LIN {X 0,Y 503.622,Z 638.337,A -85,B 0,C 180,E1 23233.198,E2 23233.198} C_VEL
LIN {X 0,Y 501.583,Z 634.122,A -85,B 0,C 180,E1 23232.199,E2 23232.199} C_VEL
LIN {X 0,Y 499.58,Z 629.914,A -85,B 0,C 180,E1 23231.195,E2 23231.195} C_VEL
LIN {X 0,Y 498.04,Z 626.665,A -85,B 0,C 180,E1 23230.41,E2 23230.41} C_VEL
LIN {X 0,Y 497.921,Z 625.951,A -85,B 0,C 180,E1 23230.237,E2 23230.237} C_VEL
LIN {X 0,Y 497.932,Z 625.949,A -85,B 0,C 180,E1 23226.688,E2 23226.688} C_VEL
LIN {X 0,Y 497.917,Z 625.952,A -85,B 0,C 180,E1 23223.108,E2 23223.108} C_VEL
LIN {X 0,Y 497.933,Z 625.957,A -85,B 0,C 180,E1 23219.54,E2 23219.54} C_VEL
LIN {X 0,Y 497.926,Z 625.949,A -85,B 0,C 180,E1 23215.854,E2 23215.854} C_VEL
LIN {X 0,Y 497.932,Z 625.949,A -85,B 0,C 180,E1 23212.268,E2 23212.268} C_VEL
LIN {X 0,Y 497.92,Z 625.957,A -85,B 0,C 180,E1 23208.65,E2 23208.65} C_VEL
LIN {X 0,Y 497.926,Z 625.958,A -85,B 0,C 180,E1 23205.106,E2 23205.106} C_VEL
LIN {X 0,Y 497.935,Z 625.96,A -85,B 0,C 180,E1 23201.502,E2 23201.502} C_VEL
LIN {X 0,Y 497.922,Z 625.959,A -85,B 0,C 180,E1 23197.943,E2 23197.943} C_VEL
LIN {X 0,Y 497.927,Z 625.957,A -85,B 0,C 180,E1 23194.294,E2 23194.294} C_VEL
LIN {X 0,Y 497.919,Z 625.959,A -85,B 0,C 180,E1 23190.792,E2 23190.792} C_VEL
LIN {X 0,Y 497.93,Z 625.957,A -85,B 0,C 180,E1 23187.283,E2 23187.283} C_VEL
LIN {X 0,Y 497.923,Z 625.955,A -85,B 0,C 180,E1 23183.815,E2 23183.815} C_VEL
LIN {X 0,Y 497.93,Z 625.956,A -85,B 0,C 180,E1 23180.27,E2 23180.27} C_VEL
LIN {X 0,Y 497.92,Z 625.916,A -85,B 0,C 180,E1 23176.628,E2 23176.628} C_VEL
LIN {X 0,Y 497.928,Z 625.947,A -85,B 0,C 180,E1 23173.056,E2 23173.056} C_VEL
LIN {X 0,Y 497.936,Z 625.963,A -85,B 0,C 180,E1 23169.533,E2 23169.533} C_VEL
LIN {X 0,Y 497.945,Z 626.094,A -85,B 0,C 180,E1 23169.367,E2 23169.367} C_VEL
LIN {X 0,Y 507.09,Z 649.982,A -85,B 0,C 180,E1 23166.816,E2 23166.816} C_VEL
LIN {X 0,Y 513.886,Z 670.595,A -85,B 0,C 180,E1 23164.716,E2 23164.716} C_VEL
LIN {X 0,Y 516.12,Z 678.989,A -85,B 0,C 180,E1 23163.912,E2 23163.912} C_VEL
LIN {X 0,Y 514.134,Z 718.892,A -85,B 0,C 180,E1 23160.89,E2 23160.89} C_VEL
LIN {X 0,Y 511.854,Z 763.473,A -85,B 0,C 180,E1 23157.516,E2 23157.516} C_VEL
LIN {X 0,Y 509.643,Z 811.319,A -85,B 0,C 180,E1 23153.959,E2 23153.959} C_VEL
LIN {X 0,Y 508.296,Z 851.099,A -85,B 0,C 180,E1 23151.154,E2 23151.154} C_VEL
LIN {X 0,Y 509.003,Z 858.968,A -85,B 0,C 180,E1 23151.003,E2 23151.003} C_VEL
LIN {X 0,Y 506.584,Z 1020.416,A -85,B 0,C 180,E1 23148.679,E2 23148.679} C_VEL
LIN {X 0,Y 506.284,Z 1037.996,A -85,B 0,C 180,E1 23148.228,E2 23148.228} C_VEL
LIN {X 0,Y 505.713,Z 1054.181,A -85,B 0,C 180,E1 23147.607,E2 23147.607} C_VEL
LIN {X 0,Y 505.321,Z 1062.229,A -85,B 0,C 180,E1 23147.218,E2 23147.218} C_VEL
LIN {X 0,Y 503.989,Z 1069.347,A -85,B 0,C 180,E1 23146.868,E2 23146.868} C_VEL
LIN {X 0,Y 497.857,Z 1084.669,A -85,B 0,C 180,E1 23146.084,E2 23146.084} C_VEL
LIN {X 0,Y 495.985,Z 1091.125,A -85,B 0,C 180,E1 23145.643,E2 23145.643} C_VEL
LIN {X 0,Y 495.757,Z 1092.898,A -85,B 0,C 180,E1 23145.5,E2 23145.5} C_VEL
LIN {X 0,Y 494.579,Z 1106.659,A -85,B 0,C 180,E1 23144.218,E2 23144.218} C_VEL
LIN {X 0,Y 493.371,Z 1119.245,A -85,B 0,C 180,E1 23142.76,E2 23142.76} C_VEL
LIN {X 0,Y 492.214,Z 1130.691,A -85,B 0,C 180,E1 23141.125,E2 23141.125} C_VEL
LIN {X 0,Y 491.214,Z 1140.574,A -85,B 0,C 180,E1 23139.37,E2 23139.37} C_VEL
LIN {X 0,Y 490.396,Z 1148.83,A -85,B 0,C 180,E1 23137.496,E2 23137.496} C_VEL
LIN {X 0,Y 489.788,Z 1155.493,A -85,B 0,C 180,E1 23135.504,E2 23135.504} C_VEL
LIN {X 0,Y 489.392,Z 1160.26,A -85,B 0,C 180,E1 23133.512,E2 23133.512} C_VEL
LIN {X 0,Y 489.172,Z 1163.258,A -85,B 0,C 180,E1 23131.521,E2 23131.521} C_VEL
LIN {X 0,Y 489.082,Z 1164.606,A -85,B 0,C 180,E1 23129.413,E2 23129.413} C_VEL
LIN {X 0,Y 489.126,Z 1164.179,A -85,B 0,C 180,E1 23127.304,E2 23127.304} C_VEL
LIN {X 0,Y 489.319,Z 1161.943,A -85,B 0,C 180,E1 23125.193,E2 23125.193} C_VEL
LIN {X 0,Y 489.663,Z 1158.025,A -85,B 0,C 180,E1 23123.197,E2 23123.197} C_VEL
LIN {X 0,Y 490.209,Z 1152.292,A -85,B 0,C 180,E1 23121.199,E2 23121.199} C_VEL
LIN {X 0,Y 490.957,Z 1145.049,A -85,B 0,C 180,E1 23119.318,E2 23119.318} C_VEL
LIN {X 0,Y 491.891,Z 1136.305,A -85,B 0,C 180,E1 23117.555,E2 23117.555} C_VEL
LIN {X 0,Y 492.983,Z 1126.106,A -85,B 0,C 180,E1 23115.912,E2 23115.912} C_VEL
LIN {X 0,Y 494.201,Z 1114.401,A -85,B 0,C 180,E1 23114.38,E2 23114.38} C_VEL
LIN {X 0,Y 495.469,Z 1101.282,A -85,B 0,C 180,E1 23112.984,E2 23112.984} C_VEL
LIN {X 0,Y 496.686,Z 1086.899,A -85,B 0,C 180,E1 23111.756,E2 23111.756} C_VEL
LIN {X 0,Y 497.789,Z 1071.409,A -85,B 0,C 180,E1 23110.704,E2 23110.704} C_VEL
LIN {X 0,Y 498.655,Z 1055.917,A -85,B 0,C 180,E1 23109.885,E2 23109.885} C_VEL
LIN {X 0,Y 499.309,Z 1038.979,A -85,B 0,C 180,E1 23109.22,E2 23109.22} C_VEL
LIN {X 0,Y 499.63,Z 1021.423,A -85,B 0,C 180,E1 23108.762,E2 23108.762} C_VEL
LIN {X 0,Y 501.594,Z 894.511,A -85,B 0,C 180,E1 23106.898,E2 23106.898} C_VEL
LIN {X 0,Y 502.065,Z 856.472,A -85,B 0,C 180,E1 23106.339,E2 23106.339} C_VEL
LIN {X 0,Y 501.456,Z 851.589,A -85,B 0,C 180,E1 23106.218,E2 23106.218} C_VEL
LIN {X 0,Y 503.183,Z 807.728,A -85,B 0,C 180,E1 23103.058,E2 23103.058} C_VEL
LIN {X 0,Y 505.515,Z 762.418,A -85,B 0,C 180,E1 23099.643,E2 23099.643} C_VEL
LIN {X 0,Y 508.171,Z 714.262,A -85,B 0,C 180,E1 23095.957,E2 23095.957} C_VEL
LIN {X 0,Y 509.871,Z 682.308,A -85,B 0,C 180,E1 23093.518,E2 23093.518} C_VEL
LIN {X 0,Y 503.228,Z 661.234,A -85,B 0,C 180,E1 23091.341,E2 23091.341} C_VEL
LIN {X 0,Y 495.525,Z 640.587,A -85,B 0,C 180,E1 23089.085,E2 23089.085} C_VEL
LIN {X 0,Y 490.002,Z 627.063,A -85,B 0,C 180,E1 23087.55,E2 23087.55} C_VEL
LIN {X 0,Y 490.019,Z 627.136,A -85,B 0,C 180,E1 23087.237,E2 23087.237} C_VEL
LIN {X 0,Y 491.489,Z 630.701,A -85,B 0,C 180,E1 23086.556,E2 23086.556} C_VEL
LIN {X 0,Y 498.257,Z 644.719,A -85,B 0,C 180,E1 23083.909,E2 23083.909} C_VEL
LIN {X 0,Y 500.365,Z 648.918,A -85,B 0,C 180,E1 23083.205,E2 23083.205} C_VEL
LIN {X 0,Y 518.762,Z 674.964,A -85,B 0,C 180,E1 23080.671,E2 23080.671} C_VEL
LIN {X 0,Y 534.168,Z 697.824,A -85,B 0,C 180,E1 23078.718,E2 23078.718} C_VEL
LIN {X 0,Y 520.026,Z 971.597,A -85,B 0,C 180,E1 23073.818,E2 23073.818} C_VEL
LIN {X 0,Y 518.593,Z 994.45,A -85,B 0,C 180,E1 23073.196,E2 23073.196} C_VEL
LIN {X 0,Y 516.689,Z 1017.478,A -85,B 0,C 180,E1 23072.37,E2 23072.37} C_VEL
LIN {X 0,Y 514.491,Z 1039.246,A -85,B 0,C 180,E1 23071.389,E2 23071.389} C_VEL
LIN {X 0,Y 512.002,Z 1059.668,A -85,B 0,C 180,E1 23070.255,E2 23070.255} C_VEL
LIN {X 0,Y 509.133,Z 1081.117,A -85,B 0,C 180,E1 23068.832,E2 23068.832} C_VEL
LIN {X 0,Y 506.332,Z 1100.244,A -85,B 0,C 180,E1 23067.331,E2 23067.331} C_VEL
LIN {X 0,Y 503.44,Z 1118.322,A -85,B 0,C 180,E1 23065.657,E2 23065.657} C_VEL
LIN {X 0,Y 500.455,Z 1136.635,A -85,B 0,C 180,E1 23063.678,E2 23063.678} C_VEL
LIN {X 0,Y 497.838,Z 1152.47,A -85,B 0,C 180,E1 23061.688,E2 23061.688} C_VEL
LIN {X 0,Y 495.417,Z 1167.155,A -85,B 0,C 180,E1 23059.516,E2 23059.516} C_VEL
LIN {X 0,Y 493.209,Z 1181.129,A -85,B 0,C 180,E1 23057.095,E2 23057.095} C_VEL
LIN {X 0,Y 491.538,Z 1192.748,A -85,B 0,C 180,E1 23054.731,E2 23054.731} C_VEL
LIN {X 0,Y 490.203,Z 1202.859,A -85,B 0,C 180,E1 23052.248,E2 23052.248} C_VEL
LIN {X 0,Y 489.216,Z 1211.985,A -85,B 0,C 180,E1 23049.529,E2 23049.529} C_VEL
LIN {X 0,Y 488.65,Z 1218.647,A -85,B 0,C 180,E1 23047.052,E2 23047.052} C_VEL
LIN {X 0,Y 488.301,Z 1223.926,A -85,B 0,C 180,E1 23044.463,E2 23044.463} C_VEL
LIN {X 0,Y 488.147,Z 1227.754,A -85,B 0,C 180,E1 23041.878,E2 23041.878} C_VEL
LIN {X 0,Y 488.091,Z 1229.852,A -85,B 0,C 180,E1 23039.413,E2 23039.413} C_VEL
LIN {X 0,Y 488.086,Z 1230.749,A -85,B 0,C 180,E1 23036.829,E2 23036.829} C_VEL
LIN {X 0,Y 488.12,Z 1230.019,A -85,B 0,C 180,E1 23034.239,E2 23034.239} C_VEL
LIN {X 0,Y 488.209,Z 1227.733,A -85,B 0,C 180,E1 23031.52,E2 23031.52} C_VEL
LIN {X 0,Y 488.421,Z 1224.179,A -85,B 0,C 180,E1 23029.024,E2 23029.024} C_VEL
LIN {X 0,Y 488.853,Z 1218.825,A -85,B 0,C 180,E1 23026.395,E2 23026.395} C_VEL
LIN {X 0,Y 489.556,Z 1212.199,A -85,B 0,C 180,E1 23023.873,E2 23023.873} C_VEL
LIN {X 0,Y 490.6,Z 1203.943,A -85,B 0,C 180,E1 23021.393,E2 23021.393} C_VEL
LIN {X 0,Y 492.129,Z 1193.445,A -85,B 0,C 180,E1 23018.798,E2 23018.798} C_VEL
LIN {X 0,Y 493.919,Z 1182.352,A -85,B 0,C 180,E1 23016.496,E2 23016.496} C_VEL
LIN {X 0,Y 496.141,Z 1169.08,A -85,B 0,C 180,E1 23014.195,E2 23014.195} C_VEL
LIN {X 0,Y 498.52,Z 1155.148,A -85,B 0,C 180,E1 23012.139,E2 23012.139} C_VEL
LIN {X 0,Y 501.101,Z 1140.099,A -85,B 0,C 180,E1 23010.228,E2 23010.228} C_VEL
LIN {X 0,Y 503.629,Z 1124.294,A -85,B 0,C 180,E1 23008.523,E2 23008.523} C_VEL
LIN {X 0,Y 506.268,Z 1106.682,A -85,B 0,C 180,E1 23006.9,E2 23006.9} C_VEL
LIN {X 0,Y 508.688,Z 1089.092,A -85,B 0,C 180,E1 23005.521,E2 23005.521} C_VEL
LIN {X 0,Y 510.84,Z 1070.657,A -85,B 0,C 180,E1 23004.318,E2 23004.318} C_VEL
LIN {X 0,Y 512.763,Z 1050.458,A -85,B 0,C 180,E1 23003.226,E2 23003.226} C_VEL
LIN {X 0,Y 514.255,Z 1030.564,A -85,B 0,C 180,E1 23002.362,E2 23002.362} C_VEL
LIN {X 0,Y 515.293,Z 1009.487,A -85,B 0,C 180,E1 23001.655,E2 23001.655} C_VEL
LIN {X 0,Y 515.797,Z 988.179,A -85,B 0,C 180,E1 23001.151,E2 23001.151} C_VEL
LIN {X 0,Y 517.226,Z 940.752,A -85,B 0,C 180,E1 23000.326,E2 23000.326} C_VEL
LIN {X 0,Y 520.642,Z 879.085,A -85,B 0,C 180,E1 22999.174,E2 22999.174} C_VEL
LIN {X 0,Y 525.552,Z 819.384,A -85,B 0,C 180,E1 22997.917,E2 22997.917} C_VEL
LIN {X 0,Y 527.75,Z 796.96,A -85,B 0,C 180,E1 22997.398,E2 22997.398} C_VEL
LIN {X 0,Y 520.311,Z 808.831,A -85,B 0,C 180,E1 22996.188,E2 22996.188} C_VEL
LIN {X 0,Y 515.367,Z 820.417,A -85,B 0,C 180,E1 22994.988,E2 22994.988} C_VEL
LIN {X 0,Y 512.446,Z 832.873,A -85,B 0,C 180,E1 22993.758,E2 22993.758} C_VEL
LIN {X 0,Y 511.546,Z 846.864,A -85,B 0,C 180,E1 22992.457,E2 22992.457} C_VEL
LIN {X 0,Y 512.945,Z 861.88,A -85,B 0,C 180,E1 22991.105,E2 22991.105} C_VEL
LIN {X 0,Y 517.01,Z 878.772,A -85,B 0,C 180,E1 22989.649,E2 22989.649} C_VEL
LIN {X 0,Y 522.772,Z 895.04,A -85,B 0,C 180,E1 22988.353,E2 22988.353} C_VEL
LIN {X 0,Y 530.728,Z 911.414,A -85,B 0,C 180,E1 22987.081,E2 22987.081} C_VEL
LIN {X 0,Y 524.079,Z 932.845,A -85,B 0,C 180,E1 22987.102,E2 22987.102} C_VEL
LIN {X 0,Y 519.267,Z 950.939,A -85,B 0,C 180,E1 22986.962,E2 22986.962} C_VEL
LIN {X 0,Y 515.69,Z 968.825,A -85,B 0,C 180,E1 22986.636,E2 22986.636} C_VEL
LIN {X 0,Y 513.389,Z 987.439,A -85,B 0,C 180,E1 22986.107,E2 22986.107} C_VEL
LIN {X 0,Y 509.621,Z 1023.418,A -85,B 0,C 180,E1 22984.852,E2 22984.852} C_VEL
LIN {X 0,Y 506.382,Z 1054.848,A -85,B 0,C 180,E1 22983.532,E2 22983.532} C_VEL
LIN {X 0,Y 503.423,Z 1085.64,A -85,B 0,C 180,E1 22981.994,E2 22981.994} C_VEL
LIN {X 0,Y 500.875,Z 1113.859,A -85,B 0,C 180,E1 22980.337,E2 22980.337} C_VEL
LIN {X 0,Y 498.595,Z 1139.721,A -85,B 0,C 180,E1 22978.575,E2 22978.575} C_VEL
LIN {X 0,Y 496.528,Z 1163.782,A -85,B 0,C 180,E1 22976.685,E2 22976.685} C_VEL
LIN {X 0,Y 494.62,Z 1185.737,A -85,B 0,C 180,E1 22974.675,E2 22974.675} C_VEL
LIN {X 0,Y 493.041,Z 1204.656,A -85,B 0,C 180,E1 22972.665,E2 22972.665} C_VEL
LIN {X 0,Y 491.658,Z 1221.239,A -85,B 0,C 180,E1 22970.601,E2 22970.601} C_VEL
LIN {X 0,Y 490.58,Z 1235.432,A -85,B 0,C 180,E1 22968.541,E2 22968.541} C_VEL
LIN {X 0,Y 489.663,Z 1248.183,A -85,B 0,C 180,E1 22966.369,E2 22966.369} C_VEL
LIN {X 0,Y 488.999,Z 1258.805,A -85,B 0,C 180,E1 22964.205,E2 22964.205} C_VEL
LIN {X 0,Y 488.554,Z 1267.998,A -85,B 0,C 180,E1 22961.931,E2 22961.931} C_VEL
LIN {X 0,Y 488.252,Z 1275.736,A -85,B 0,C 180,E1 22959.55,E2 22959.55} C_VEL
LIN {X 0,Y 488.122,Z 1281.616,A -85,B 0,C 180,E1 22957.18,E2 22957.18} C_VEL
LIN {X 0,Y 488.072,Z 1285.747,A -85,B 0,C 180,E1 22954.82,E2 22954.82} C_VEL
LIN {X 0,Y 488.064,Z 1288.404,A -85,B 0,C 180,E1 22952.35,E2 22952.35} C_VEL
LIN {X 0,Y 488.082,Z 1289.345,A -85,B 0,C 180,E1 22950.002,E2 22950.002} C_VEL
LIN {X 0,Y 488.042,Z 1288.685,A -85,B 0,C 180,E1 22947.536,E2 22947.536} C_VEL
LIN {X 0,Y 488.033,Z 1286.434,A -85,B 0,C 180,E1 22945.065,E2 22945.065} C_VEL
LIN {X 0,Y 488.072,Z 1282.457,A -85,B 0,C 180,E1 22942.548,E2 22942.548} C_VEL
LIN {X 0,Y 488.237,Z 1276.355,A -85,B 0,C 180,E1 22939.858,E2 22939.858} C_VEL
LIN {X 0,Y 488.608,Z 1268.875,A -85,B 0,C 180,E1 22937.354,E2 22937.354} C_VEL
LIN {X 0,Y 489.31,Z 1258.996,A -85,B 0,C 180,E1 22934.692,E2 22934.692} C_VEL
LIN {X 0,Y 490.393,Z 1247.083,A -85,B 0,C 180,E1 22932.07,E2 22932.07} C_VEL
LIN {X 0,Y 491.81,Z 1234.099,A -85,B 0,C 180,E1 22929.658,E2 22929.658} C_VEL
LIN {X 0,Y 493.701,Z 1218.912,A -85,B 0,C 180,E1 22927.245,E2 22927.245} C_VEL
LIN {X 0,Y 496.134,Z 1201.151,A -85,B 0,C 180,E1 22924.836,E2 22924.836} C_VEL
LIN {X 0,Y 498.818,Z 1182.632,A -85,B 0,C 180,E1 22922.677,E2 22922.677} C_VEL
LIN {X 0,Y 501.889,Z 1162.559,A -85,B 0,C 180,E1 22920.656,E2 22920.656} C_VEL
LIN {X 0,Y 505.491,Z 1139.288,A -85,B 0,C 180,E1 22918.655,E2 22918.655} C_VEL
LIN {X 0,Y 508.695,Z 1118.909,A -85,B 0,C 180,E1 22917.148,E2 22917.148} C_VEL
LIN {X 0,Y 512.451,Z 1094.537,A -85,B 0,C 180,E1 22915.609,E2 22915.609} C_VEL
LIN {X 0,Y 515.778,Z 1072.564,A -85,B 0,C 180,E1 22914.441,E2 22914.441} C_VEL
LIN {X 0,Y 519.332,Z 1047.797,A -85,B 0,C 180,E1 22913.358,E2 22913.358} C_VEL
LIN {X 0,Y 522.293,Z 1025.669,A -85,B 0,C 180,E1 22912.57,E2 22912.57} C_VEL
LIN {X 0,Y 525.245,Z 999.637,A -85,B 0,C 180,E1 22911.846,E2 22911.846} C_VEL
LIN {X 0,Y 527.354,Z 975.274,A -85,B 0,C 180,E1 22911.33,E2 22911.33} C_VEL
LIN {X 0,Y 530.154,Z 954.931,A -85,B 0,C 180,E1 22911.079,E2 22911.079} C_VEL
LIN {X 0,Y 532.607,Z 942.044,A -85,B 0,C 180,E1 22910.963,E2 22910.963} C_VEL
LIN {X 0,Y 536.49,Z 935.316,A -85,B 0,C 180,E1 22910.582,E2 22910.582} C_VEL
LIN {X 0,Y 529.21,Z 920.705,A -85,B 0,C 180,E1 22908.748,E2 22908.748} C_VEL
LIN {X 0,Y 523.75,Z 904.487,A -85,B 0,C 180,E1 22906.826,E2 22906.826} C_VEL
LIN {X 0,Y 520.425,Z 886.754,A -85,B 0,C 180,E1 22904.839,E2 22904.839} C_VEL
LIN {X 0,Y 519.332,Z 867.376,A -85,B 0,C 180,E1 22902.816,E2 22902.816} C_VEL
LIN {X 0,Y 520.601,Z 845.317,A -85,B 0,C 180,E1 22900.657,E2 22900.657} C_VEL
LIN {X 0,Y 525.45,Z 806.808,A -85,B 0,C 180,E1 22897.047,E2 22897.047} C_VEL
LIN {X 0,Y 530.041,Z 771.847,A -85,B 0,C 180,E1 22893.708,E2 22893.708} C_VEL
LIN {X 0,Y 534.385,Z 739.455,A -85,B 0,C 180,E1 22890.537,E2 22890.537} C_VEL
LIN {X 0,Y 535.607,Z 729.994,A -85,B 0,C 180,E1 22889.589,E2 22889.589} C_VEL
LIN {X 0,Y 527.935,Z 710.743,A -85,B 0,C 180,E1 22886.429,E2 22886.429} C_VEL
LIN {X 0,Y 520.037,Z 692,A -85,B 0,C 180,E1 22883.094,E2 22883.094} C_VEL
LIN {X 0,Y 512.802,Z 675.646,A -85,B 0,C 180,E1 22879.952,E2 22879.952} C_VEL
LIN {X 0,Y 506.279,Z 661.298,A -85,B 0,C 180,E1 22876.996,E2 22876.996} C_VEL
LIN {X 0,Y 499.858,Z 647.869,A -85,B 0,C 180,E1 22874.007,E2 22874.007} C_VEL
LIN {X 0,Y 495.726,Z 639.359,A -85,B 0,C 180,E1 22871.991,E2 22871.991} C_VEL
LIN {X 0,Y 493.67,Z 635.137,A -85,B 0,C 180,E1 22870.976,E2 22870.976} C_VEL
LIN {X 0,Y 491.719,Z 630.999,A -85,B 0,C 180,E1 22869.953,E2 22869.953} C_VEL
LIN {X 0,Y 490.138,Z 627.802,A -85,B 0,C 180,E1 22869.132,E2 22869.132} C_VEL
LIN {X 0,Y 489.988,Z 626.938,A -85,B 0,C 180,E1 22868.922,E2 22868.922} C_VEL
LIN {X 0,Y 489.995,Z 626.939,A -85,B 0,C 180,E1 22865.386,E2 22865.386} C_VEL
LIN {X 0,Y 489.994,Z 626.938,A -85,B 0,C 180,E1 22861.637,E2 22861.637} C_VEL
LIN {X 0,Y 489.979,Z 626.939,A -85,B 0,C 180,E1 22858.012,E2 22858.012} C_VEL
LIN {X 0,Y 489.989,Z 626.946,A -85,B 0,C 180,E1 22854.379,E2 22854.379} C_VEL
LIN {X 0,Y 489.984,Z 626.945,A -85,B 0,C 180,E1 22850.841,E2 22850.841} C_VEL
LIN {X 0,Y 489.992,Z 626.94,A -85,B 0,C 180,E1 22847.259,E2 22847.259} C_VEL
LIN {X 0,Y 489.984,Z 626.938,A -85,B 0,C 180,E1 22843.644,E2 22843.644} C_VEL
LIN {X 0,Y 489.991,Z 626.937,A -85,B 0,C 180,E1 22840.075,E2 22840.075} C_VEL
LIN {X 0,Y 489.989,Z 626.936,A -85,B 0,C 180,E1 22836.551,E2 22836.551} C_VEL
LIN {X 0,Y 489.98,Z 626.934,A -85,B 0,C 180,E1 22833.062,E2 22833.062} C_VEL
LIN {X 0,Y 489.985,Z 626.938,A -85,B 0,C 180,E1 22829.597,E2 22829.597} C_VEL
LIN {X 0,Y 489.996,Z 626.938,A -85,B 0,C 180,E1 22825.94,E2 22825.94} C_VEL
LIN {X 0,Y 489.997,Z 626.939,A -85,B 0,C 180,E1 22822.252,E2 22822.252} C_VEL
LIN {X 0,Y 489.985,Z 626.939,A -85,B 0,C 180,E1 22818.61,E2 22818.61} C_VEL
LIN {X 0,Y 489.981,Z 626.924,A -85,B 0,C 180,E1 22815.078,E2 22815.078} C_VEL
LIN {X 0,Y 489.998,Z 626.914,A -85,B 0,C 180,E1 22811.504,E2 22811.504} C_VEL
LIN {X 0,Y 489.986,Z 626.981,A -85,B 0,C 180,E1 22809.95,E2 22809.95} C_VEL
LIN {X 0,Y 498.827,Z 649.766,A -85,B 0,C 180,E1 22807.46,E2 22807.46} C_VEL
LIN {X 0,Y 505.699,Z 669.989,A -85,B 0,C 180,E1 22805.352,E2 22805.352} C_VEL
LIN {X 0,Y 508.926,Z 681.63,A -85,B 0,C 180,E1 22804.193,E2 22804.193} C_VEL
LIN {X 0,Y 506.912,Z 721.32,A -85,B 0,C 180,E1 22801.181,E2 22801.181} C_VEL
LIN {X 0,Y 504.446,Z 767.454,A -85,B 0,C 180,E1 22797.664,E2 22797.664} C_VEL
LIN {X 0,Y 502.253,Z 813.696,A -85,B 0,C 180,E1 22794.209,E2 22794.209} C_VEL
LIN {X 0,Y 500.918,Z 852.144,A -85,B 0,C 180,E1 22791.488,E2 22791.488} C_VEL
LIN {X 0,Y 501.594,Z 859.853,A -85,B 0,C 180,E1 22791.338,E2 22791.338} C_VEL
LIN {X 0,Y 499.074,Z 1021.09,A -85,B 0,C 180,E1 22788.985,E2 22788.985} C_VEL
LIN {X 0,Y 498.765,Z 1038.703,A -85,B 0,C 180,E1 22788.529,E2 22788.529} C_VEL
LIN {X 0,Y 498.157,Z 1055.322,A -85,B 0,C 180,E1 22787.883,E2 22787.883} C_VEL
LIN {X 0,Y 497.267,Z 1071.796,A -85,B 0,C 180,E1 22787.01,E2 22787.01} C_VEL
LIN {X 0,Y 496.21,Z 1087.141,A -85,B 0,C 180,E1 22785.963,E2 22785.963} C_VEL
LIN {X 0,Y 495.757,Z 1092.898,A -85,B 0,C 180,E1 22785.5,E2 22785.5} C_VEL
LIN {X 0,Y 494.313,Z 1099.187,A -85,B 0,C 180,E1 22784.998,E2 22784.998} C_VEL
LIN {X 0,Y 488.294,Z 1111.875,A -85,B 0,C 180,E1 22783.925,E2 22783.925} C_VEL
LIN {X 0,Y 485.952,Z 1118.163,A -85,B 0,C 180,E1 22783.24,E2 22783.24} C_VEL
LIN {X 0,Y 485.702,Z 1119.657,A -85,B 0,C 180,E1 22783.048,E2 22783.048} C_VEL
LIN {X 0,Y 484.479,Z 1131.231,A -85,B 0,C 180,E1 22781.382,E2 22781.382} C_VEL
LIN {X 0,Y 483.443,Z 1140.967,A -85,B 0,C 180,E1 22779.642,E2 22779.642} C_VEL
LIN {X 0,Y 482.619,Z 1148.928,A -85,B 0,C 180,E1 22777.857,E2 22777.857} C_VEL
LIN {X 0,Y 481.944,Z 1155.798,A -85,B 0,C 180,E1 22775.833,E2 22775.833} C_VEL
LIN {X 0,Y 481.501,Z 1160.747,A -85,B 0,C 180,E1 22773.809,E2 22773.809} C_VEL
LIN {X 0,Y 481.244,Z 1164.101,A -85,B 0,C 180,E1 22771.665,E2 22771.665} C_VEL
LIN {X 0,Y 481.141,Z 1165.539,A -85,B 0,C 180,E1 22769.522,E2 22769.522} C_VEL
LIN {X 0,Y 481.18,Z 1165.191,A -85,B 0,C 180,E1 22767.378,E2 22767.378} C_VEL
LIN {X 0,Y 481.378,Z 1163.056,A -85,B 0,C 180,E1 22765.232,E2 22765.232} C_VEL
LIN {X 0,Y 481.735,Z 1159.243,A -85,B 0,C 180,E1 22763.204,E2 22763.204} C_VEL
LIN {X 0,Y 482.299,Z 1153.599,A -85,B 0,C 180,E1 22761.174,E2 22761.174} C_VEL
LIN {X 0,Y 483.073,Z 1146.453,A -85,B 0,C 180,E1 22759.262,E2 22759.262} C_VEL
LIN {X 0,Y 484.045,Z 1137.864,A -85,B 0,C 180,E1 22757.472,E2 22757.472} C_VEL
LIN {X 0,Y 485.175,Z 1127.799,A -85,B 0,C 180,E1 22755.802,E2 22755.802} C_VEL
LIN {X 0,Y 486.426,Z 1116.308,A -85,B 0,C 180,E1 22754.255,E2 22754.255} C_VEL
LIN {X 0,Y 487.772,Z 1102.991,A -85,B 0,C 180,E1 22752.797,E2 22752.797} C_VEL
LIN {X 0,Y 489.019,Z 1089.166,A -85,B 0,C 180,E1 22751.575,E2 22751.575} C_VEL
LIN {X 0,Y 490.152,Z 1074.106,A -85,B 0,C 180,E1 22750.515,E2 22750.515} C_VEL
LIN {X 0,Y 491.113,Z 1057.858,A -85,B 0,C 180,E1 22749.624,E2 22749.624} C_VEL
LIN {X 0,Y 491.826,Z 1040.688,A -85,B 0,C 180,E1 22748.926,E2 22748.926} C_VEL
LIN {X 0,Y 492.179,Z 1023.103,A -85,B 0,C 180,E1 22748.451,E2 22748.451} C_VEL
LIN {X 0,Y 493.142,Z 956.489,A -85,B 0,C 180,E1 22747.44,E2 22747.44} C_VEL
LIN {X 0,Y 494.737,Z 857.413,A -85,B 0,C 180,E1 22745.979,E2 22745.979} C_VEL
LIN {X 0,Y 494.122,Z 852.727,A -85,B 0,C 180,E1 22745.872,E2 22745.872} C_VEL
LIN {X 0,Y 495.912,Z 808.893,A -85,B 0,C 180,E1 22742.695,E2 22742.695} C_VEL
LIN {X 0,Y 498.439,Z 761.451,A -85,B 0,C 180,E1 22739.098,E2 22739.098} C_VEL
LIN {X 0,Y 501.032,Z 716.223,A -85,B 0,C 180,E1 22735.612,E2 22735.612} C_VEL
LIN {X 0,Y 502.686,Z 684.816,A -85,B 0,C 180,E1 22733.189,E2 22733.189} C_VEL
LIN {X 0,Y 496.087,Z 663.92,A -85,B 0,C 180,E1 22730.996,E2 22730.996} C_VEL
LIN {X 0,Y 488.626,Z 644.049,A -85,B 0,C 180,E1 22728.781,E2 22728.781} C_VEL
LIN {X 0,Y 483.86,Z 632.705,A -85,B 0,C 180,E1 22727.447,E2 22727.447} C_VEL
LIN {X 0,Y 484.494,Z 633.594,A -85,B 0,C 180,E1 22727.234,E2 22727.234} C_VEL
LIN {X 0,Y 488.84,Z 642.71,A -85,B 0,C 180,E1 22725.444,E2 22725.444} C_VEL
LIN {X 0,Y 492.891,Z 650.929,A -85,B 0,C 180,E1 22723.952,E2 22723.952} C_VEL
LIN {X 0,Y 509.541,Z 674.266,A -85,B 0,C 180,E1 22721.59,E2 22721.59} C_VEL
LIN {X 0,Y 527.777,Z 701.194,A -85,B 0,C 180,E1 22719.212,E2 22719.212} C_VEL
LIN {X 0,Y 513.091,Z 972.818,A -85,B 0,C 180,E1 22714.247,E2 22714.247} C_VEL
LIN {X 0,Y 511.606,Z 995.57,A -85,B 0,C 180,E1 22713.615,E2 22713.615} C_VEL
LIN {X 0,Y 509.588,Z 1019.037,A -85,B 0,C 180,E1 22712.756,E2 22712.756} C_VEL
LIN {X 0,Y 507.297,Z 1040.818,A -85,B 0,C 180,E1 22711.753,E2 22711.753} C_VEL
LIN {X 0,Y 504.62,Z 1062.025,A -85,B 0,C 180,E1 22710.547,E2 22710.547} C_VEL
LIN {X 0,Y 501.663,Z 1083.244,A -85,B 0,C 180,E1 22709.1,E2 22709.1} C_VEL
LIN {X 0,Y 498.8,Z 1102.102,A -85,B 0,C 180,E1 22707.585,E2 22707.585} C_VEL
LIN {X 0,Y 495.845,Z 1119.99,A -85,B 0,C 180,E1 22705.892,E2 22705.892} C_VEL
LIN {X 0,Y 492.857,Z 1137.708,A -85,B 0,C 180,E1 22703.938,E2 22703.938} C_VEL
LIN {X 0,Y 490.158,Z 1153.483,A -85,B 0,C 180,E1 22701.92,E2 22701.92} C_VEL
LIN {X 0,Y 487.719,Z 1167.75,A -85,B 0,C 180,E1 22699.772,E2 22699.772} C_VEL
LIN {X 0,Y 485.476,Z 1181.418,A -85,B 0,C 180,E1 22697.376,E2 22697.376} C_VEL
LIN {X 0,Y 483.73,Z 1193.079,A -85,B 0,C 180,E1 22694.974,E2 22694.974} C_VEL
LIN {X 0,Y 482.334,Z 1203.244,A -85,B 0,C 180,E1 22692.45,E2 22692.45} C_VEL
LIN {X 0,Y 481.33,Z 1212.062,A -85,B 0,C 180,E1 22689.808,E2 22689.808} C_VEL
LIN {X 0,Y 480.717,Z 1218.789,A -85,B 0,C 180,E1 22687.289,E2 22687.289} C_VEL
LIN {X 0,Y 480.341,Z 1224.189,A -85,B 0,C 180,E1 22684.657,E2 22684.657} C_VEL
LIN {X 0,Y 480.172,Z 1227.924,A -85,B 0,C 180,E1 22682.148,E2 22682.148} C_VEL
LIN {X 0,Y 480.109,Z 1230.276,A -85,B 0,C 180,E1 22679.523,E2 22679.523} C_VEL
LIN {X 0,Y 480.097,Z 1231.213,A -85,B 0,C 180,E1 22677.015,E2 22677.015} C_VEL
LIN {X 0,Y 480.135,Z 1230.643,A -85,B 0,C 180,E1 22674.383,E2 22674.383} C_VEL
LIN {X 0,Y 480.235,Z 1228.673,A -85,B 0,C 180,E1 22671.74,E2 22671.74} C_VEL
LIN {X 0,Y 480.439,Z 1225.257,A -85,B 0,C 180,E1 22669.204,E2 22669.204} C_VEL
LIN {X 0,Y 480.902,Z 1219.89,A -85,B 0,C 180,E1 22666.411,E2 22666.411} C_VEL
LIN {X 0,Y 481.634,Z 1213.404,A -85,B 0,C 180,E1 22663.848,E2 22663.848} C_VEL
LIN {X 0,Y 482.751,Z 1205.116,A -85,B 0,C 180,E1 22661.274,E2 22661.274} C_VEL
LIN {X 0,Y 484.406,Z 1194.477,A -85,B 0,C 180,E1 22658.57,E2 22658.57} C_VEL
LIN {X 0,Y 486.331,Z 1183.278,A -85,B 0,C 180,E1 22656.195,E2 22656.195} C_VEL
LIN {X 0,Y 488.634,Z 1170.308,A -85,B 0,C 180,E1 22653.899,E2 22653.899} C_VEL
LIN {X 0,Y 491.136,Z 1156.503,A -85,B 0,C 180,E1 22651.815,E2 22651.815} C_VEL
LIN {X 0,Y 493.869,Z 1141.433,A -85,B 0,C 180,E1 22649.861,E2 22649.861} C_VEL
LIN {X 0,Y 496.542,Z 1125.633,A -85,B 0,C 180,E1 22648.123,E2 22648.123} C_VEL
LIN {X 0,Y 499.366,Z 1107.798,A -85,B 0,C 180,E1 22646.451,E2 22646.451} C_VEL
LIN {X 0,Y 501.901,Z 1090.265,A -85,B 0,C 180,E1 22645.057,E2 22645.057} C_VEL
LIN {X 0,Y 504.219,Z 1071.547,A -85,B 0,C 180,E1 22643.815,E2 22643.815} C_VEL
LIN {X 0,Y 506.188,Z 1051.875,A -85,B 0,C 180,E1 22642.739,E2 22642.739} C_VEL
LIN {X 0,Y 507.819,Z 1030.954,A -85,B 0,C 180,E1 22641.824,E2 22641.824} C_VEL
LIN {X 0,Y 508.901,Z 1010.034,A -85,B 0,C 180,E1 22641.118,E2 22641.118} C_VEL
LIN {X 0,Y 509.482,Z 988.003,A -85,B 0,C 180,E1 22640.593,E2 22640.593} C_VEL
LIN {X 0,Y 511.1,Z 943.871,A -85,B 0,C 180,E1 22639.785,E2 22639.785} C_VEL
LIN {X 0,Y 514.851,Z 886.81,A -85,B 0,C 180,E1 22638.657,E2 22638.657} C_VEL
LIN {X 0,Y 520.188,Z 831.257,A -85,B 0,C 180,E1 22637.426,E2 22637.426} C_VEL
LIN {X 0,Y 522.286,Z 812.776,A -85,B 0,C 180,E1 22636.978,E2 22636.978} C_VEL
LIN {X 0,Y 515.703,Z 824.644,A -85,B 0,C 180,E1 22635.761,E2 22635.761} C_VEL
LIN {X 0,Y 511.393,Z 836.851,A -85,B 0,C 180,E1 22634.544,E2 22634.544} C_VEL
LIN {X 0,Y 509.165,Z 849.897,A -85,B 0,C 180,E1 22633.285,E2 22633.285} C_VEL
LIN {X 0,Y 509.135,Z 863.894,A -85,B 0,C 180,E1 22631.962,E2 22631.962} C_VEL
LIN {X 0,Y 511.46,Z 878.475,A -85,B 0,C 180,E1 22630.609,E2 22630.609} C_VEL
LIN {X 0,Y 516.141,Z 895.312,A -85,B 0,C 180,E1 22629.184,E2 22629.184} C_VEL
LIN {X 0,Y 522.983,Z 911.283,A -85,B 0,C 180,E1 22627.85,E2 22627.85} C_VEL
LIN {X 0,Y 523.902,Z 913.41,A -85,B 0,C 180,E1 22627.693,E2 22627.693} C_VEL
LIN {X 0,Y 516.737,Z 937.023,A -85,B 0,C 180,E1 22627.671,E2 22627.671} C_VEL
LIN {X 0,Y 512.295,Z 954.451,A -85,B 0,C 180,E1 22627.482,E2 22627.482} C_VEL
LIN {X 0,Y 508.877,Z 972.315,A -85,B 0,C 180,E1 22627.107,E2 22627.107} C_VEL
LIN {X 0,Y 505.673,Z 998.578,A -85,B 0,C 180,E1 22626.263,E2 22626.263} C_VEL
LIN {X 0,Y 501.664,Z 1033.434,A -85,B 0,C 180,E1 22624.928,E2 22624.928} C_VEL
LIN {X 0,Y 498.309,Z 1064.666,A -85,B 0,C 180,E1 22623.492,E2 22623.492} C_VEL
LIN {X 0,Y 495.274,Z 1094.694,A -85,B 0,C 180,E1 22621.867,E2 22621.867} C_VEL
LIN {X 0,Y 492.589,Z 1122.767,A -85,B 0,C 180,E1 22620.092,E2 22620.092} C_VEL
LIN {X 0,Y 490.096,Z 1149.677,A -85,B 0,C 180,E1 22618.119,E2 22618.119} C_VEL
LIN {X 0,Y 488.104,Z 1171.53,A -85,B 0,C 180,E1 22616.264,E2 22616.264} C_VEL
LIN {X 0,Y 486.263,Z 1192.367,A -85,B 0,C 180,E1 22614.22,E2 22614.22} C_VEL
LIN {X 0,Y 484.696,Z 1210.286,A -85,B 0,C 180,E1 22612.181,E2 22612.181} C_VEL
LIN {X 0,Y 483.365,Z 1226.043,A -85,B 0,C 180,E1 22610.085,E2 22610.085} C_VEL
LIN {X 0,Y 482.248,Z 1240.235,A -85,B 0,C 180,E1 22607.872,E2 22607.872} C_VEL
LIN {X 0,Y 481.421,Z 1252.183,A -85,B 0,C 180,E1 22605.666,E2 22605.666} C_VEL
LIN {X 0,Y 480.802,Z 1262.564,A -85,B 0,C 180,E1 22603.348,E2 22603.348} C_VEL
LIN {X 0,Y 480.395,Z 1271.396,A -85,B 0,C 180,E1 22600.92,E2 22600.92} C_VEL
LIN {X 0,Y 480.186,Z 1278.375,A -85,B 0,C 180,E1 22598.469,E2 22598.469} C_VEL
LIN {X 0,Y 480.099,Z 1283.522,A -85,B 0,C 180,E1 22595.979,E2 22595.979} C_VEL
LIN {X 0,Y 480.079,Z 1286.971,A -85,B 0,C 180,E1 22593.464,E2 22593.464} C_VEL
LIN {X 0,Y 480.085,Z 1288.613,A -85,B 0,C 180,E1 22591.076,E2 22591.076} C_VEL
LIN {X 0,Y 480.067,Z 1288.656,A -85,B 0,C 180,E1 22588.569,E2 22588.569} C_VEL
LIN {X 0,Y 480.047,Z 1287.081,A -85,B 0,C 180,E1 22586.06,E2 22586.06} C_VEL
LIN {X 0,Y 480.05,Z 1283.83,A -85,B 0,C 180,E1 22583.544,E2 22583.544} C_VEL
LIN {X 0,Y 480.146,Z 1278.645,A -85,B 0,C 180,E1 22580.895,E2 22580.895} C_VEL
LIN {X 0,Y 480.428,Z 1271.944,A -85,B 0,C 180,E1 22578.355,E2 22578.355} C_VEL
LIN {X 0,Y 481.013,Z 1262.776,A -85,B 0,C 180,E1 22575.624,E2 22575.624} C_VEL
LIN {X 0,Y 481.887,Z 1252.426,A -85,B 0,C 180,E1 22573.115,E2 22573.115} C_VEL
LIN {X 0,Y 483.224,Z 1239.807,A -85,B 0,C 180,E1 22570.542,E2 22570.542} C_VEL
LIN {X 0,Y 485.061,Z 1224.813,A -85,B 0,C 180,E1 22567.967,E2 22567.967} C_VEL
LIN {X 0,Y 487.215,Z 1208.983,A -85,B 0,C 180,E1 22565.64,E2 22565.64} C_VEL
LIN {X 0,Y 489.808,Z 1191.352,A -85,B 0,C 180,E1 22563.398,E2 22563.398} C_VEL
LIN {X 0,Y 493.018,Z 1170.719,A -85,B 0,C 180,E1 22561.141,E2 22561.141} C_VEL
LIN {X 0,Y 496.294,Z 1150.156,A -85,B 0,C 180,E1 22559.223,E2 22559.223} C_VEL
LIN {X 0,Y 499.72,Z 1129.083,A -85,B 0,C 180,E1 22557.506,E2 22557.506} C_VEL
LIN {X 0,Y 503.384,Z 1106.368,A -85,B 0,C 180,E1 22555.937,E2 22555.937} C_VEL
LIN {X 0,Y 507.067,Z 1083.359,A -85,B 0,C 180,E1 22554.57,E2 22554.57} C_VEL
LIN {X 0,Y 510.605,Z 1059.918,A -85,B 0,C 180,E1 22553.424,E2 22553.424} C_VEL
LIN {X 0,Y 514.156,Z 1035.566,A -85,B 0,C 180,E1 22552.437,E2 22552.437} C_VEL
LIN {X 0,Y 517.294,Z 1011.342,A -85,B 0,C 180,E1 22551.672,E2 22551.672} C_VEL
LIN {X 0,Y 519.905,Z 985.089,A -85,B 0,C 180,E1 22551.016,E2 22551.016} C_VEL
LIN {X 0,Y 522.057,Z 965.13,A -85,B 0,C 180,E1 22550.677,E2 22550.677} C_VEL
LIN {X 0,Y 526.207,Z 941.269,A -85,B 0,C 180,E1 22550.449,E2 22550.449} C_VEL
LIN {X 0,Y 528.296,Z 937.077,A -85,B 0,C 180,E1 22550.232,E2 22550.232} C_VEL
LIN {X 0,Y 521.05,Z 921.552,A -85,B 0,C 180,E1 22548.287,E2 22548.287} C_VEL
LIN {X 0,Y 515.923,Z 904.797,A -85,B 0,C 180,E1 22546.294,E2 22546.294} C_VEL
LIN {X 0,Y 513.043,Z 887.28,A -85,B 0,C 180,E1 22544.338,E2 22544.338} C_VEL
LIN {X 0,Y 512.31,Z 867.487,A -85,B 0,C 180,E1 22542.258,E2 22542.258} C_VEL
LIN {X 0,Y 513.874,Z 845.366,A -85,B 0,C 180,E1 22540.095,E2 22540.095} C_VEL
LIN {X 0,Y 518.737,Z 808.42,A -85,B 0,C 180,E1 22536.594,E2 22536.594} C_VEL
LIN {X 0,Y 523.488,Z 773.701,A -85,B 0,C 180,E1 22533.243,E2 22533.243} C_VEL
LIN {X 0,Y 528.052,Z 740.77,A -85,B 0,C 180,E1 22529.993,E2 22529.993} C_VEL
LIN {X 0,Y 529.02,Z 733.979,A -85,B 0,C 180,E1 22529.31,E2 22529.31} C_VEL
LIN {X 0,Y 521.519,Z 715.037,A -85,B 0,C 180,E1 22526.166,E2 22526.166} C_VEL
LIN {X 0,Y 513.87,Z 696.818,A -85,B 0,C 180,E1 22522.902,E2 22522.902} C_VEL
LIN {X 0,Y 506.677,Z 680.445,A -85,B 0,C 180,E1 22519.732,E2 22519.732} C_VEL
LIN {X 0,Y 500.294,Z 666.388,A -85,B 0,C 180,E1 22516.806,E2 22516.806} C_VEL
LIN {X 0,Y 494.233,Z 653.536,A -85,B 0,C 180,E1 22513.931,E2 22513.931} C_VEL
LIN {X 0,Y 489.832,Z 644.525,A -85,B 0,C 180,E1 22511.779,E2 22511.779} C_VEL
LIN {X 0,Y 487.787,Z 640.338,A -85,B 0,C 180,E1 22510.751,E2 22510.751} C_VEL
LIN {X 0,Y 486.005,Z 636.492,A -85,B 0,C 180,E1 22509.791,E2 22509.791} C_VEL
LIN {X 0,Y 484.274,Z 632.685,A -85,B 0,C 180,E1 22508.848,E2 22508.848} C_VEL
LIN {X 0,Y 482.293,Z 629.087,A -85,B 0,C 180,E1 22507.865,E2 22507.865} C_VEL
LIN {X 0,Y 482.049,Z 627.932,A -85,B 0,C 180,E1 22507.569,E2 22507.569} C_VEL
LIN {X 0,Y 482.039,Z 627.928,A -85,B 0,C 180,E1 22504.044,E2 22504.044} C_VEL
LIN {X 0,Y 482.056,Z 627.927,A -85,B 0,C 180,E1 22500.475,E2 22500.475} C_VEL
LIN {X 0,Y 482.041,Z 627.937,A -85,B 0,C 180,E1 22496.908,E2 22496.908} C_VEL
LIN {X 0,Y 482.059,Z 627.926,A -85,B 0,C 180,E1 22493.21,E2 22493.21} C_VEL
LIN {X 0,Y 482.047,Z 627.925,A -85,B 0,C 180,E1 22489.603,E2 22489.603} C_VEL
LIN {X 0,Y 482.058,Z 627.927,A -85,B 0,C 180,E1 22485.955,E2 22485.955} C_VEL
LIN {X 0,Y 482.042,Z 627.934,A -85,B 0,C 180,E1 22482.371,E2 22482.371} C_VEL
LIN {X 0,Y 482.05,Z 627.933,A -85,B 0,C 180,E1 22478.843,E2 22478.843} C_VEL
LIN {X 0,Y 482.056,Z 627.933,A -85,B 0,C 180,E1 22475.098,E2 22475.098} C_VEL
LIN {X 0,Y 482.056,Z 627.935,A -85,B 0,C 180,E1 22471.37,E2 22471.37} C_VEL
LIN {X 0,Y 482.043,Z 627.933,A -85,B 0,C 180,E1 22467.785,E2 22467.785} C_VEL
LIN {X 0,Y 482.049,Z 627.926,A -85,B 0,C 180,E1 22464.193,E2 22464.193} C_VEL
LIN {X 0,Y 482.057,Z 627.927,A -85,B 0,C 180,E1 22460.601,E2 22460.601} C_VEL
LIN {X 0,Y 482.042,Z 627.894,A -85,B 0,C 180,E1 22457.07,E2 22457.07} C_VEL
LIN {X 0,Y 482.051,Z 627.93,A -85,B 0,C 180,E1 22453.357,E2 22453.357} C_VEL
LIN {X 0,Y 482.074,Z 628.052,A -85,B 0,C 180,E1 22450.541,E2 22450.541} C_VEL
LIN {X 0,Y 491.269,Z 651.393,A -85,B 0,C 180,E1 22447.925,E2 22447.925} C_VEL
LIN {X 0,Y 498.097,Z 671.275,A -85,B 0,C 180,E1 22445.806,E2 22445.806} C_VEL
LIN {X 0,Y 501.836,Z 683.814,A -85,B 0,C 180,E1 22444.536,E2 22444.536} C_VEL
LIN {X 0,Y 499.427,Z 728.654,A -85,B 0,C 180,E1 22441.098,E2 22441.098} C_VEL
LIN {X 0,Y 496.776,Z 776.579,A -85,B 0,C 180,E1 22437.423,E2 22437.423} C_VEL
LIN {X 0,Y 494.42,Z 827.068,A -85,B 0,C 180,E1 22433.666,E2 22433.666} C_VEL
LIN {X 0,Y 493.563,Z 853.224,A -85,B 0,C 180,E1 22431.832,E2 22431.832} C_VEL
LIN {X 0,Y 494.205,Z 860.683,A -85,B 0,C 180,E1 22431.684,E2 22431.684} C_VEL
LIN {X 0,Y 491.58,Z 1021.795,A -85,B 0,C 180,E1 22429.301,E2 22429.301} C_VEL
LIN {X 0,Y 491.263,Z 1039.31,A -85,B 0,C 180,E1 22428.843,E2 22428.843} C_VEL
LIN {X 0,Y 490.68,Z 1055.225,A -85,B 0,C 180,E1 22428.226,E2 22428.226} C_VEL
LIN {X 0,Y 489.81,Z 1071.067,A -85,B 0,C 180,E1 22427.393,E2 22427.393} C_VEL
LIN {X 0,Y 488.727,Z 1086.422,A -85,B 0,C 180,E1 22426.355,E2 22426.355} C_VEL
LIN {X 0,Y 487.551,Z 1100.57,A -85,B 0,C 180,E1 22425.156,E2 22425.156} C_VEL
LIN {X 0,Y 486.322,Z 1113.571,A -85,B 0,C 180,E1 22423.796,E2 22423.796} C_VEL
LIN {X 0,Y 485.702,Z 1119.657,A -85,B 0,C 180,E1 22423.048,E2 22423.048} C_VEL
LIN {X 0,Y 484.199,Z 1124.9,A -85,B 0,C 180,E1 22422.384,E2 22422.384} C_VEL
LIN {X 0,Y 478.167,Z 1135.243,A -85,B 0,C 180,E1 22420.985,E2 22420.985} C_VEL
LIN {X 0,Y 475.903,Z 1140.216,A -85,B 0,C 180,E1 22420.148,E2 22420.148} C_VEL
LIN {X 0,Y 475.683,Z 1141.361,A -85,B 0,C 180,E1 22419.923,E2 22419.923} C_VEL
LIN {X 0,Y 474.754,Z 1149.921,A -85,B 0,C 180,E1 22417.988,E2 22417.988} C_VEL
LIN {X 0,Y 474.044,Z 1156.78,A -85,B 0,C 180,E1 22415.931,E2 22415.931} C_VEL
LIN {X 0,Y 473.578,Z 1161.72,A -85,B 0,C 180,E1 22413.872,E2 22413.872} C_VEL
LIN {X 0,Y 473.307,Z 1165.065,A -85,B 0,C 180,E1 22411.693,E2 22411.693} C_VEL
LIN {X 0,Y 473.197,Z 1166.493,A -85,B 0,C 180,E1 22409.514,E2 22409.514} C_VEL
LIN {X 0,Y 473.241,Z 1166.138,A -85,B 0,C 180,E1 22407.334,E2 22407.334} C_VEL
LIN {X 0,Y 473.453,Z 1163.995,A -85,B 0,C 180,E1 22405.153,E2 22405.153} C_VEL
LIN {X 0,Y 473.833,Z 1160.171,A -85,B 0,C 180,E1 22403.09,E2 22403.09} C_VEL
LIN {X 0,Y 474.431,Z 1154.519,A -85,B 0,C 180,E1 22401.026,E2 22401.026} C_VEL
LIN {X 0,Y 475.25,Z 1147.362,A -85,B 0,C 180,E1 22399.083,E2 22399.083} C_VEL
LIN {X 0,Y 476.273,Z 1138.759,A -85,B 0,C 180,E1 22397.264,E2 22397.264} C_VEL
LIN {X 0,Y 477.458,Z 1128.678,A -85,B 0,C 180,E1 22395.568,E2 22395.568} C_VEL
LIN {X 0,Y 478.767,Z 1117.17,A -85,B 0,C 180,E1 22393.996,E2 22393.996} C_VEL
LIN {X 0,Y 480.14,Z 1104.144,A -85,B 0,C 180,E1 22392.548,E2 22392.548} C_VEL
LIN {X 0,Y 481.399,Z 1090.82,A -85,B 0,C 180,E1 22391.344,E2 22391.344} C_VEL
LIN {X 0,Y 482.586,Z 1075.839,A -85,B 0,C 180,E1 22390.26,E2 22390.26} C_VEL
LIN {X 0,Y 483.583,Z 1059.801,A -85,B 0,C 180,E1 22389.356,E2 22389.356} C_VEL
LIN {X 0,Y 484.336,Z 1042.704,A -85,B 0,C 180,E1 22388.637,E2 22388.637} C_VEL
LIN {X 0,Y 484.741,Z 1025.349,A -85,B 0,C 180,E1 22388.143,E2 22388.143} C_VEL
LIN {X 0,Y 485.314,Z 981.118,A -85,B 0,C 180,E1 22387.442,E2 22387.442} C_VEL
LIN {X 0,Y 487.429,Z 858.359,A -85,B 0,C 180,E1 22385.608,E2 22385.608} C_VEL
LIN {X 0,Y 486.817,Z 853.448,A -85,B 0,C 180,E1 22385.486,E2 22385.486} C_VEL
LIN {X 0,Y 488.713,Z 809.281,A -85,B 0,C 180,E1 22382.259,E2 22382.259} C_VEL
LIN {X 0,Y 491.287,Z 763.173,A -85,B 0,C 180,E1 22378.734,E2 22378.734} C_VEL
LIN {X 0,Y 494.082,Z 715.749,A -85,B 0,C 180,E1 22375.059,E2 22375.059} C_VEL
LIN {X 0,Y 495.543,Z 687.383,A -85,B 0,C 180,E1 22372.847,E2 22372.847} C_VEL
LIN {X 0,Y 488.951,Z 666.553,A -85,B 0,C 180,E1 22370.624,E2 22370.624} C_VEL
LIN {X 0,Y 481.411,Z 646.456,A -85,B 0,C 180,E1 22368.344,E2 22368.344} C_VEL
LIN {X 0,Y 478.322,Z 639.11,A -85,B 0,C 180,E1 22367.448,E2 22367.448} C_VEL
LIN {X 0,Y 478.99,Z 639.656,A -85,B 0,C 180,E1 22367.277,E2 22367.277} C_VEL
LIN {X 0,Y 483.109,Z 648.134,A -85,B 0,C 180,E1 22365.607,E2 22365.607} C_VEL
LIN {X 0,Y 485.586,Z 653.07,A -85,B 0,C 180,E1 22364.71,E2 22364.71} C_VEL
LIN {X 0,Y 501.456,Z 675.168,A -85,B 0,C 180,E1 22362.393,E2 22362.393} C_VEL
LIN {X 0,Y 520.009,Z 702.414,A -85,B 0,C 180,E1 22359.895,E2 22359.895} C_VEL
LIN {X 0,Y 521.416,Z 704.929,A -85,B 0,C 180,E1 22359.704,E2 22359.704} C_VEL
LIN {X 0,Y 506.2,Z 973.181,A -85,B 0,C 180,E1 22354.703,E2 22354.703} C_VEL
LIN {X 0,Y 504.662,Z 996.162,A -85,B 0,C 180,E1 22354.058,E2 22354.058} C_VEL
LIN {X 0,Y 502.669,Z 1018.799,A -85,B 0,C 180,E1 22353.224,E2 22353.224} C_VEL
LIN {X 0,Y 500.254,Z 1041.158,A -85,B 0,C 180,E1 22352.186,E2 22352.186} C_VEL
LIN {X 0,Y 497.494,Z 1062.417,A -85,B 0,C 180,E1 22350.966,E2 22350.966} C_VEL
LIN {X 0,Y 494.563,Z 1082.912,A -85,B 0,C 180,E1 22349.559,E2 22349.559} C_VEL
LIN {X 0,Y 491.601,Z 1101.918,A -85,B 0,C 180,E1 22348.024,E2 22348.024} C_VEL
LIN {X 0,Y 488.52,Z 1119.995,A -85,B 0,C 180,E1 22346.298,E2 22346.298} C_VEL
LIN {X 0,Y 485.346,Z 1138.216,A -85,B 0,C 180,E1 22344.268,E2 22344.268} C_VEL
LIN {X 0,Y 482.632,Z 1153.57,A -85,B 0,C 180,E1 22342.28,E2 22342.28} C_VEL
LIN {X 0,Y 480.035,Z 1168.266,A -85,B 0,C 180,E1 22340.045,E2 22340.045} C_VEL
LIN {X 0,Y 477.652,Z 1182.302,A -85,B 0,C 180,E1 22337.544,E2 22337.544} C_VEL
LIN {X 0,Y 475.851,Z 1193.93,A -85,B 0,C 180,E1 22335.103,E2 22335.103} C_VEL
LIN {X 0,Y 474.408,Z 1204.042,A -85,B 0,C 180,E1 22332.538,E2 22332.538} C_VEL
LIN {X 0,Y 473.334,Z 1213.155,A -85,B 0,C 180,E1 22329.729,E2 22329.729} C_VEL
LIN {X 0,Y 472.698,Z 1220.108,A -85,B 0,C 180,E1 22327.047,E2 22327.047} C_VEL
LIN {X 0,Y 472.331,Z 1225.261,A -85,B 0,C 180,E1 22324.371,E2 22324.371} C_VEL
LIN {X 0,Y 472.17,Z 1228.958,A -85,B 0,C 180,E1 22321.699,E2 22321.699} C_VEL
LIN {X 0,Y 472.116,Z 1230.984,A -85,B 0,C 180,E1 22319.151,E2 22319.151} C_VEL
LIN {X 0,Y 472.123,Z 1231.708,A -85,B 0,C 180,E1 22316.357,E2 22316.357} C_VEL
LIN {X 0,Y 472.167,Z 1230.927,A -85,B 0,C 180,E1 22313.8,E2 22313.8} C_VEL
LIN {X 0,Y 472.286,Z 1228.612,A -85,B 0,C 180,E1 22311.109,E2 22311.109} C_VEL
LIN {X 0,Y 472.59,Z 1224.836,A -85,B 0,C 180,E1 22308.405,E2 22308.405} C_VEL
LIN {X 0,Y 473.136,Z 1219.297,A -85,B 0,C 180,E1 22305.685,E2 22305.685} C_VEL
LIN {X 0,Y 474.052,Z 1212.08,A -85,B 0,C 180,E1 22302.951,E2 22302.951} C_VEL
LIN {X 0,Y 475.376,Z 1203.501,A -85,B 0,C 180,E1 22300.334,E2 22300.334} C_VEL
LIN {X 0,Y 477.076,Z 1193.405,A -85,B 0,C 180,E1 22297.836,E2 22297.836} C_VEL
LIN {X 0,Y 479.291,Z 1181.373,A -85,B 0,C 180,E1 22295.34,E2 22295.34} C_VEL
LIN {X 0,Y 481.744,Z 1168.635,A -85,B 0,C 180,E1 22293.097,E2 22293.097} C_VEL
LIN {X 0,Y 484.651,Z 1153.558,A -85,B 0,C 180,E1 22290.863,E2 22290.863} C_VEL
LIN {X 0,Y 487.478,Z 1138.332,A -85,B 0,C 180,E1 22288.951,E2 22288.951} C_VEL
LIN {X 0,Y 490.52,Z 1121.28,A -85,B 0,C 180,E1 22287.124,E2 22287.124} C_VEL
LIN {X 0,Y 493.34,Z 1104.173,A -85,B 0,C 180,E1 22285.565,E2 22285.565} C_VEL
LIN {X 0,Y 495.886,Z 1086.486,A -85,B 0,C 180,E1 22284.215,E2 22284.215} C_VEL
LIN {X 0,Y 498.262,Z 1067.32,A -85,B 0,C 180,E1 22282.985,E2 22282.985} C_VEL
LIN {X 0,Y 500.187,Z 1048.732,A -85,B 0,C 180,E1 22281.997,E2 22281.997} C_VEL
LIN {X 0,Y 501.794,Z 1027.762,A -85,B 0,C 180,E1 22281.116,E2 22281.116} C_VEL
LIN {X 0,Y 502.801,Z 1006.755,A -85,B 0,C 180,E1 22280.446,E2 22280.446} C_VEL
LIN {X 0,Y 503.58,Z 978.937,A -85,B 0,C 180,E1 22279.832,E2 22279.832} C_VEL
LIN {X 0,Y 506.521,Z 927.976,A -85,B 0,C 180,E1 22278.826,E2 22278.826} C_VEL
LIN {X 0,Y 511.099,Z 876.915,A -85,B 0,C 180,E1 22277.707,E2 22277.707} C_VEL
LIN {X 0,Y 517.039,Z 828.705,A -85,B 0,C 180,E1 22276.547,E2 22276.547} C_VEL
LIN {X 0,Y 511.161,Z 841.061,A -85,B 0,C 180,E1 22275.322,E2 22275.322} C_VEL
LIN {X 0,Y 507.554,Z 853.629,A -85,B 0,C 180,E1 22274.081,E2 22274.081} C_VEL
LIN {X 0,Y 506.155,Z 866.376,A -85,B 0,C 180,E1 22272.828,E2 22272.828} C_VEL
LIN {X 0,Y 506.939,Z 879.658,A -85,B 0,C 180,E1 22271.528,E2 22271.528} C_VEL
LIN {X 0,Y 510.087,Z 895.348,A -85,B 0,C 180,E1 22270.094,E2 22270.094} C_VEL
LIN {X 0,Y 515.36,Z 910.643,A -85,B 0,C 180,E1 22268.744,E2 22268.744} C_VEL
LIN {X 0,Y 517.368,Z 915.528,A -85,B 0,C 180,E1 22268.336,E2 22268.336} C_VEL
LIN {X 0,Y 510.383,Z 938.84,A -85,B 0,C 180,E1 22268.286,E2 22268.286} C_VEL
LIN {X 0,Y 505.818,Z 956.983,A -85,B 0,C 180,E1 22268.048,E2 22268.048} C_VEL
LIN {X 0,Y 502.462,Z 974.44,A -85,B 0,C 180,E1 22267.638,E2 22267.638} C_VEL
LIN {X 0,Y 498.549,Z 1004.644,A -85,B 0,C 180,E1 22266.597,E2 22266.597} C_VEL
LIN {X 0,Y 494.154,Z 1039.862,A -85,B 0,C 180,E1 22265.148,E2 22265.148} C_VEL
LIN {X 0,Y 490.536,Z 1071.28,A -85,B 0,C 180,E1 22263.603,E2 22263.603} C_VEL
LIN {X 0,Y 487.458,Z 1099.974,A -85,B 0,C 180,E1 22261.954,E2 22261.954} C_VEL
LIN {X 0,Y 484.642,Z 1127.982,A -85,B 0,C 180,E1 22260.09,E2 22260.09} C_VEL
LIN {X 0,Y 482.114,Z 1153.94,A -85,B 0,C 180,E1 22258.087,E2 22258.087} C_VEL
LIN {X 0,Y 479.999,Z 1175.991,A -85,B 0,C 180,E1 22256.126,E2 22256.126} C_VEL
LIN {X 0,Y 478.123,Z 1195.949,A -85,B 0,C 180,E1 22254.068,E2 22254.068} C_VEL
LIN {X 0,Y 476.546,Z 1213.553,A -85,B 0,C 180,E1 22251.965,E2 22251.965} C_VEL
LIN {X 0,Y 475.215,Z 1229.058,A -85,B 0,C 180,E1 22249.803,E2 22249.803} C_VEL
LIN {X 0,Y 474.125,Z 1242.506,A -85,B 0,C 180,E1 22247.592,E2 22247.592} C_VEL
LIN {X 0,Y 473.317,Z 1254.201,A -85,B 0,C 180,E1 22245.313,E2 22245.313} C_VEL
LIN {X 0,Y 472.714,Z 1264.23,A -85,B 0,C 180,E1 22242.958,E2 22242.958} C_VEL
LIN {X 0,Y 472.362,Z 1272.257,A -85,B 0,C 180,E1 22240.614,E2 22240.614} C_VEL
LIN {X 0,Y 472.166,Z 1278.814,A -85,B 0,C 180,E1 22238.158,E2 22238.158} C_VEL
LIN {X 0,Y 472.098,Z 1283.6,A -85,B 0,C 180,E1 22235.715,E2 22235.715} C_VEL
LIN {X 0,Y 472.096,Z 1286.703,A -85,B 0,C 180,E1 22233.28,E2 22233.28} C_VEL
LIN {X 0,Y 472.096,Z 1288.206,A -85,B 0,C 180,E1 22230.73,E2 22230.73} C_VEL
LIN {X 0,Y 472.083,Z 1288.042,A -85,B 0,C 180,E1 22228.181,E2 22228.181} C_VEL
LIN {X 0,Y 472.055,Z 1286.3,A -85,B 0,C 180,E1 22225.75,E2 22225.75} C_VEL
LIN {X 0,Y 472.063,Z 1282.83,A -85,B 0,C 180,E1 22223.19,E2 22223.19} C_VEL
LIN {X 0,Y 472.175,Z 1277.714,A -85,B 0,C 180,E1 22220.617,E2 22220.617} C_VEL
LIN {X 0,Y 472.489,Z 1270.818,A -85,B 0,C 180,E1 22218.032,E2 22218.032} C_VEL
LIN {X 0,Y 473.101,Z 1261.674,A -85,B 0,C 180,E1 22215.31,E2 22215.31} C_VEL
LIN {X 0,Y 474.124,Z 1250.331,A -85,B 0,C 180,E1 22212.576,E2 22212.576} C_VEL
LIN {X 0,Y 475.516,Z 1237.776,A -85,B 0,C 180,E1 22210.04,E2 22210.04} C_VEL
LIN {X 0,Y 477.466,Z 1222.671,A -85,B 0,C 180,E1 22207.448,E2 22207.448} C_VEL
LIN {X 0,Y 480.012,Z 1204.862,A -85,B 0,C 180,E1 22204.855,E2 22204.855} C_VEL
LIN {X 0,Y 483.001,Z 1185.533,A -85,B 0,C 180,E1 22202.456,E2 22202.456} C_VEL
LIN {X 0,Y 486.294,Z 1165.264,A -85,B 0,C 180,E1 22200.298,E2 22200.298} C_VEL
LIN {X 0,Y 489.572,Z 1145.468,A -85,B 0,C 180,E1 22198.479,E2 22198.479} C_VEL
LIN {X 0,Y 493.495,Z 1122.141,A -85,B 0,C 180,E1 22196.629,E2 22196.629} C_VEL
LIN {X 0,Y 496.966,Z 1101.476,A -85,B 0,C 180,E1 22195.224,E2 22195.224} C_VEL
LIN {X 0,Y 501.002,Z 1076.624,A -85,B 0,C 180,E1 22193.792,E2 22193.792} C_VEL
LIN {X 0,Y 504.68,Z 1053.417,A -85,B 0,C 180,E1 22192.683,E2 22192.683} C_VEL
LIN {X 0,Y 508.347,Z 1028.299,A -85,B 0,C 180,E1 22191.717,E2 22191.717} C_VEL
LIN {X 0,Y 511.637,Z 1002.888,A -85,B 0,C 180,E1 22190.939,E2 22190.939} C_VEL
LIN {X 0,Y 513.994,Z 978.056,A -85,B 0,C 180,E1 22190.364,E2 22190.364} C_VEL
LIN {X 0,Y 516.76,Z 957.498,A -85,B 0,C 180,E1 22190.068,E2 22190.068} C_VEL
LIN {X 0,Y 520.253,Z 938.983,A -85,B 0,C 180,E1 22189.901,E2 22189.901} C_VEL
LIN {X 0,Y 513.278,Z 923.224,A -85,B 0,C 180,E1 22187.92,E2 22187.92} C_VEL
LIN {X 0,Y 508.369,Z 906.061,A -85,B 0,C 180,E1 22185.875,E2 22185.875} C_VEL
LIN {X 0,Y 505.716,Z 887.673,A -85,B 0,C 180,E1 22183.811,E2 22183.811} C_VEL
LIN {X 0,Y 505.315,Z 867.315,A -85,B 0,C 180,E1 22181.672,E2 22181.672} C_VEL
LIN {X 0,Y 507.392,Z 844.028,A -85,B 0,C 180,E1 22179.387,E2 22179.387} C_VEL
LIN {X 0,Y 512.24,Z 808.454,A -85,B 0,C 180,E1 22175.984,E2 22175.984} C_VEL
LIN {X 0,Y 517.097,Z 774.258,A -85,B 0,C 180,E1 22172.649,E2 22172.649} C_VEL
LIN {X 0,Y 521.85,Z 741.457,A -85,B 0,C 180,E1 22169.374,E2 22169.374} C_VEL
LIN {X 0,Y 522.302,Z 737.552,A -85,B 0,C 180,E1 22168.969,E2 22168.969} C_VEL
LIN {X 0,Y 514.534,Z 718.004,A -85,B 0,C 180,E1 22165.681,E2 22165.681} C_VEL
LIN {X 0,Y 507.438,Z 701.038,A -85,B 0,C 180,E1 22162.597,E2 22162.597} C_VEL
LIN {X 0,Y 500.522,Z 685.15,A -85,B 0,C 180,E1 22159.488,E2 22159.488} C_VEL
LIN {X 0,Y 494.23,Z 671.315,A -85,B 0,C 180,E1 22156.575,E2 22156.575} C_VEL
LIN {X 0,Y 488.354,Z 658.743,A -85,B 0,C 180,E1 22153.739,E2 22153.739} C_VEL
LIN {X 0,Y 482.695,Z 646.753,A -85,B 0,C 180,E1 22150.866,E2 22150.866} C_VEL
LIN {X 0,Y 479.909,Z 641.41,A -85,B 0,C 180,E1 22149.474,E2 22149.474} C_VEL
LIN {X 0,Y 477.949,Z 637.302,A -85,B 0,C 180,E1 22148.421,E2 22148.421} C_VEL
LIN {X 0,Y 476.09,Z 633.277,A -85,B 0,C 180,E1 22147.361,E2 22147.361} C_VEL
LIN {X 0,Y 474.279,Z 629.857,A -85,B 0,C 180,E1 22146.415,E2 22146.415} C_VEL
LIN {X 0,Y 474.102,Z 628.914,A -85,B 0,C 180,E1 22146.175,E2 22146.175} C_VEL
LIN {X 0,Y 474.111,Z 628.924,A -85,B 0,C 180,E1 22142.538,E2 22142.538} C_VEL
LIN {X 0,Y 474.117,Z 628.915,A -85,B 0,C 180,E1 22138.912,E2 22138.912} C_VEL
LIN {X 0,Y 474.107,Z 628.916,A -85,B 0,C 180,E1 22135.161,E2 22135.161} C_VEL
LIN {X 0,Y 474.102,Z 628.924,A -85,B 0,C 180,E1 22131.632,E2 22131.632} C_VEL
LIN {X 0,Y 474.116,Z 628.925,A -85,B 0,C 180,E1 22127.949,E2 22127.949} C_VEL
LIN {X 0,Y 474.107,Z 628.921,A -85,B 0,C 180,E1 22124.339,E2 22124.339} C_VEL
LIN {X 0,Y 474.116,Z 628.918,A -85,B 0,C 180,E1 22120.664,E2 22120.664} C_VEL
LIN {X 0,Y 474.103,Z 628.917,A -85,B 0,C 180,E1 22117.035,E2 22117.035} C_VEL
LIN {X 0,Y 474.112,Z 628.913,A -85,B 0,C 180,E1 22113.401,E2 22113.401} C_VEL
LIN {X 0,Y 474.105,Z 628.917,A -85,B 0,C 180,E1 22109.843,E2 22109.843} C_VEL
LIN {X 0,Y 474.116,Z 628.919,A -85,B 0,C 180,E1 22106.167,E2 22106.167} C_VEL
LIN {X 0,Y 474.116,Z 628.92,A -85,B 0,C 180,E1 22102.447,E2 22102.447} C_VEL
LIN {X 0,Y 474.119,Z 628.918,A -85,B 0,C 180,E1 22098.838,E2 22098.838} C_VEL
LIN {X 0,Y 474.104,Z 628.897,A -85,B 0,C 180,E1 22095.12,E2 22095.12} C_VEL
LIN {X 0,Y 474.119,Z 628.89,A -85,B 0,C 180,E1 22091.466,E2 22091.466} C_VEL
LIN {X 0,Y 474.131,Z 629.097,A -85,B 0,C 180,E1 22091.16,E2 22091.16} C_VEL
LIN {X 0,Y 483.408,Z 652.182,A -85,B 0,C 180,E1 22088.503,E2 22088.503} C_VEL
LIN {X 0,Y 490.527,Z 672.647,A -85,B 0,C 180,E1 22086.274,E2 22086.274} C_VEL
LIN {X 0,Y 494.679,Z 686.741,A -85,B 0,C 180,E1 22084.819,E2 22084.819} C_VEL
LIN {X 0,Y 492.355,Z 728.592,A -85,B 0,C 180,E1 22081.595,E2 22081.595} C_VEL
LIN {X 0,Y 489.648,Z 775.907,A -85,B 0,C 180,E1 22077.945,E2 22077.945} C_VEL
LIN {X 0,Y 487.319,Z 822.885,A -85,B 0,C 180,E1 22074.411,E2 22074.411} C_VEL
LIN {X 0,Y 486.192,Z 854.046,A -85,B 0,C 180,E1 22072.192,E2 22072.192} C_VEL
LIN {X 0,Y 486.832,Z 861.597,A -85,B 0,C 180,E1 22072.04,E2 22072.04} C_VEL
LIN {X 0,Y 484.098,Z 1022.623,A -85,B 0,C 180,E1 22069.623,E2 22069.623} C_VEL
LIN {X 0,Y 483.767,Z 1040.268,A -85,B 0,C 180,E1 22069.156,E2 22069.156} C_VEL
LIN {X 0,Y 483.151,Z 1056.373,A -85,B 0,C 180,E1 22068.52,E2 22068.52} C_VEL
LIN {X 0,Y 482.255,Z 1072.075,A -85,B 0,C 180,E1 22067.681,E2 22067.681} C_VEL
LIN {X 0,Y 481.105,Z 1087.73,A -85,B 0,C 180,E1 22066.603,E2 22066.603} C_VEL
LIN {X 0,Y 479.842,Z 1102.267,A -85,B 0,C 180,E1 22065.344,E2 22065.344} C_VEL
LIN {X 0,Y 478.621,Z 1114.604,A -85,B 0,C 180,E1 22064.023,E2 22064.023} C_VEL
LIN {X 0,Y 477.341,Z 1126.493,A -85,B 0,C 180,E1 22062.458,E2 22062.458} C_VEL
LIN {X 0,Y 476.107,Z 1137.588,A -85,B 0,C 180,E1 22060.648,E2 22060.648} C_VEL
LIN {X 0,Y 475.683,Z 1141.361,A -85,B 0,C 180,E1 22059.923,E2 22059.923} C_VEL
LIN {X 0,Y 474.288,Z 1145.364,A -85,B 0,C 180,E1 22059.137,E2 22059.137} C_VEL
LIN {X 0,Y 468.855,Z 1152.603,A -85,B 0,C 180,E1 22057.581,E2 22057.581} C_VEL
LIN {X 0,Y 466.531,Z 1156.078,A -85,B 0,C 180,E1 22056.617,E2 22056.617} C_VEL
LIN {X 0,Y 466.207,Z 1157.206,A -85,B 0,C 180,E1 22056.233,E2 22056.233} C_VEL
LIN {X 0,Y 465.702,Z 1162.207,A -85,B 0,C 180,E1 22054.185,E2 22054.185} C_VEL
LIN {X 0,Y 465.384,Z 1165.729,A -85,B 0,C 180,E1 22051.968,E2 22051.968} C_VEL
LIN {X 0,Y 465.26,Z 1167.404,A -85,B 0,C 180,E1 22049.752,E2 22049.752} C_VEL
LIN {X 0,Y 465.289,Z 1167.214,A -85,B 0,C 180,E1 22047.535,E2 22047.535} C_VEL
LIN {X 0,Y 465.49,Z 1165.241,A -85,B 0,C 180,E1 22045.316,E2 22045.316} C_VEL
LIN {X 0,Y 465.875,Z 1161.66,A -85,B 0,C 180,E1 22043.219,E2 22043.219} C_VEL
LIN {X 0,Y 466.479,Z 1156.215,A -85,B 0,C 180,E1 22041.12,E2 22041.12} C_VEL
LIN {X 0,Y 467.367,Z 1148.767,A -85,B 0,C 180,E1 22039.022,E2 22039.022} C_VEL
LIN {X 0,Y 468.424,Z 1140.28,A -85,B 0,C 180,E1 22037.172,E2 22037.172} C_VEL
LIN {X 0,Y 469.655,Z 1130.373,A -85,B 0,C 180,E1 22035.449,E2 22035.449} C_VEL
LIN {X 0,Y 471.007,Z 1119.013,A -85,B 0,C 180,E1 22033.852,E2 22033.852} C_VEL
LIN {X 0,Y 472.487,Z 1105.575,A -85,B 0,C 180,E1 22032.32,E2 22032.32} C_VEL
LIN {X 0,Y 473.863,Z 1091.635,A -85,B 0,C 180,E1 22031.036,E2 22031.036} C_VEL
LIN {X 0,Y 475.097,Z 1076.607,A -85,B 0,C 180,E1 22029.936,E2 22029.936} C_VEL
LIN {X 0,Y 476.135,Z 1060.516,A -85,B 0,C 180,E1 22029.018,E2 22029.018} C_VEL
LIN {X 0,Y 476.913,Z 1043.437,A -85,B 0,C 180,E1 22028.292,E2 22028.292} C_VEL
LIN {X 0,Y 477.329,Z 1026.207,A -85,B 0,C 180,E1 22027.797,E2 22027.797} C_VEL
LIN {X 0,Y 477.925,Z 981.89,A -85,B 0,C 180,E1 22027.083,E2 22027.083} C_VEL
LIN {X 0,Y 480.141,Z 859.307,A -85,B 0,C 180,E1 22025.227,E2 22025.227} C_VEL
LIN {X 0,Y 479.544,Z 854.215,A -85,B 0,C 180,E1 22025.089,E2 22025.089} C_VEL
LIN {X 0,Y 481.502,Z 810.525,A -85,B 0,C 180,E1 22021.874,E2 22021.874} C_VEL
LIN {X 0,Y 484.171,Z 764.076,A -85,B 0,C 180,E1 22018.304,E2 22018.304} C_VEL
LIN {X 0,Y 487.019,Z 717.849,A -85,B 0,C 180,E1 22014.693,E2 22014.693} C_VEL
LIN {X 0,Y 488.585,Z 690.583,A -85,B 0,C 180,E1 22012.565,E2 22012.565} C_VEL
LIN {X 0,Y 482.247,Z 670.403,A -85,B 0,C 180,E1 22010.378,E2 22010.378} C_VEL
LIN {X 0,Y 475.04,Z 651.03,A -85,B 0,C 180,E1 22008.144,E2 22008.144} C_VEL
LIN {X 0,Y 472.811,Z 645.529,A -85,B 0,C 180,E1 22007.451,E2 22007.451} C_VEL
LIN {X 0,Y 473.86,Z 646.263,A -85,B 0,C 180,E1 22007.198,E2 22007.198} C_VEL
LIN {X 0,Y 478.329,Z 655.231,A -85,B 0,C 180,E1 22005.486,E2 22005.486} C_VEL
LIN {X 0,Y 494.45,Z 677.767,A -85,B 0,C 180,E1 22003.047,E2 22003.047} C_VEL
LIN {X 0,Y 511.667,Z 702.838,A -85,B 0,C 180,E1 22000.67,E2 22000.67} C_VEL
LIN {X 0,Y 515.065,Z 708.361,A -85,B 0,C 180,E1 22000.211,E2 22000.211} C_VEL
LIN {X 0,Y 499.291,Z 974.125,A -85,B 0,C 180,E1 21995.153,E2 21995.153} C_VEL
LIN {X 0,Y 497.716,Z 996.883,A -85,B 0,C 180,E1 21994.504,E2 21994.504} C_VEL
LIN {X 0,Y 495.663,Z 1019.54,A -85,B 0,C 180,E1 21993.659,E2 21993.659} C_VEL
LIN {X 0,Y 493.367,Z 1040.18,A -85,B 0,C 180,E1 21992.691,E2 21992.691} C_VEL
LIN {X 0,Y 490.65,Z 1060.813,A -85,B 0,C 180,E1 21991.515,E2 21991.515} C_VEL
LIN {X 0,Y 487.738,Z 1080.937,A -85,B 0,C 180,E1 21990.15,E2 21990.15} C_VEL
LIN {X 0,Y 484.635,Z 1100.158,A -85,B 0,C 180,E1 21988.598,E2 21988.598} C_VEL
LIN {X 0,Y 481.351,Z 1119.191,A -85,B 0,C 180,E1 21986.793,E2 21986.793} C_VEL
LIN {X 0,Y 478.213,Z 1136.716,A -85,B 0,C 180,E1 21984.852,E2 21984.852} C_VEL
LIN {X 0,Y 475.282,Z 1152.714,A -85,B 0,C 180,E1 21982.774,E2 21982.774} C_VEL
LIN {X 0,Y 472.607,Z 1167.32,A -85,B 0,C 180,E1 21980.561,E2 21980.561} C_VEL
LIN {X 0,Y 470.274,Z 1180.665,A -85,B 0,C 180,E1 21978.213,E2 21978.213} C_VEL
LIN {X 0,Y 468.305,Z 1192.517,A -85,B 0,C 180,E1 21975.733,E2 21975.733} C_VEL
LIN {X 0,Y 466.738,Z 1203.029,A -85,B 0,C 180,E1 21973.126,E2 21973.126} C_VEL
LIN {X 0,Y 465.626,Z 1211.785,A -85,B 0,C 180,E1 21970.517,E2 21970.517} C_VEL
LIN {X 0,Y 464.866,Z 1219.037,A -85,B 0,C 180,E1 21967.788,E2 21967.788} C_VEL
LIN {X 0,Y 464.412,Z 1224.899,A -85,B 0,C 180,E1 21964.941,E2 21964.941} C_VEL
LIN {X 0,Y 464.213,Z 1228.711,A -85,B 0,C 180,E1 21962.346,E2 21962.346} C_VEL
LIN {X 0,Y 464.138,Z 1231.267,A -85,B 0,C 180,E1 21959.506,E2 21959.506} C_VEL
LIN {X 0,Y 464.13,Z 1232.228,A -85,B 0,C 180,E1 21956.913,E2 21956.913} C_VEL
LIN {X 0,Y 464.18,Z 1231.68,A -85,B 0,C 180,E1 21954.189,E2 21954.189} C_VEL
LIN {X 0,Y 464.297,Z 1229.72,A -85,B 0,C 180,E1 21951.454,E2 21951.454} C_VEL
LIN {X 0,Y 464.558,Z 1226.329,A -85,B 0,C 180,E1 21948.83,E2 21948.83} C_VEL
LIN {X 0,Y 465.126,Z 1220.967,A -85,B 0,C 180,E1 21945.941,E2 21945.941} C_VEL
LIN {X 0,Y 466.001,Z 1214.52,A -85,B 0,C 180,E1 21943.29,E2 21943.29} C_VEL
LIN {X 0,Y 467.299,Z 1206.242,A -85,B 0,C 180,E1 21940.631,E2 21940.631} C_VEL
LIN {X 0,Y 469.106,Z 1196.152,A -85,B 0,C 180,E1 21937.967,E2 21937.967} C_VEL
LIN {X 0,Y 471.259,Z 1185.177,A -85,B 0,C 180,E1 21935.539,E2 21935.539} C_VEL
LIN {X 0,Y 473.854,Z 1172.256,A -85,B 0,C 180,E1 21933.156,E2 21933.156} C_VEL
LIN {X 0,Y 476.822,Z 1157.734,A -85,B 0,C 180,E1 21930.889,E2 21930.889} C_VEL
LIN {X 0,Y 479.94,Z 1142.219,A -85,B 0,C 180,E1 21928.832,E2 21928.832} C_VEL
LIN {X 0,Y 483.141,Z 1125.501,A -85,B 0,C 180,E1 21926.949,E2 21926.949} C_VEL
LIN {X 0,Y 486.129,Z 1108.357,A -85,B 0,C 180,E1 21925.329,E2 21925.329} C_VEL
LIN {X 0,Y 488.982,Z 1090.18,A -85,B 0,C 180,E1 21923.874,E2 21923.874} C_VEL
LIN {X 0,Y 491.429,Z 1072.425,A -85,B 0,C 180,E1 21922.675,E2 21922.675} C_VEL
LIN {X 0,Y 493.604,Z 1053.04,A -85,B 0,C 180,E1 21921.596,E2 21921.596} C_VEL
LIN {X 0,Y 495.349,Z 1032.765,A -85,B 0,C 180,E1 21920.695,E2 21920.695} C_VEL
LIN {X 0,Y 496.567,Z 1011.694,A -85,B 0,C 180,E1 21919.971,E2 21919.971} C_VEL
LIN {X 0,Y 497.534,Z 984.282,A -85,B 0,C 180,E1 21919.31,E2 21919.31} C_VEL
LIN {X 0,Y 500.313,Z 941.055,A -85,B 0,C 180,E1 21918.403,E2 21918.403} C_VEL
LIN {X 0,Y 505.143,Z 893.264,A -85,B 0,C 180,E1 21917.311,E2 21917.311} C_VEL
LIN {X 0,Y 511.857,Z 845.267,A -85,B 0,C 180,E1 21916.1,E2 21916.1} C_VEL
LIN {X 0,Y 506.766,Z 857.706,A -85,B 0,C 180,E1 21914.869,E2 21914.869} C_VEL
LIN {X 0,Y 504.03,Z 869.657,A -85,B 0,C 180,E1 21913.66,E2 21913.66} C_VEL
LIN {X 0,Y 503.394,Z 881.978,A -85,B 0,C 180,E1 21912.397,E2 21912.397} C_VEL
LIN {X 0,Y 504.872,Z 895.552,A -85,B 0,C 180,E1 21911.056,E2 21911.056} C_VEL
LIN {X 0,Y 508.44,Z 909.825,A -85,B 0,C 180,E1 21909.723,E2 21909.723} C_VEL
LIN {X 0,Y 511.17,Z 917.741,A -85,B 0,C 180,E1 21909.015,E2 21909.015} C_VEL
LIN {X 0,Y 504.628,Z 939.627,A -85,B 0,C 180,E1 21908.943,E2 21908.943} C_VEL
LIN {X 0,Y 499.98,Z 958.145,A -85,B 0,C 180,E1 21908.68,E2 21908.68} C_VEL
LIN {X 0,Y 496.489,Z 975.689,A -85,B 0,C 180,E1 21908.239,E2 21908.239} C_VEL
LIN {X 0,Y 491.851,Z 1008.468,A -85,B 0,C 180,E1 21907.042,E2 21907.042} C_VEL
LIN {X 0,Y 487.259,Z 1042.233,A -85,B 0,C 180,E1 21905.576,E2 21905.576} C_VEL
LIN {X 0,Y 483.289,Z 1074.029,A -85,B 0,C 180,E1 21903.938,E2 21903.938} C_VEL
LIN {X 0,Y 479.894,Z 1103.504,A -85,B 0,C 180,E1 21902.166,E2 21902.166} C_VEL
LIN {X 0,Y 476.789,Z 1132.438,A -85,B 0,C 180,E1 21900.151,E2 21900.151} C_VEL
LIN {X 0,Y 474.195,Z 1157.577,A -85,B 0,C 180,E1 21898.118,E2 21898.118} C_VEL
LIN {X 0,Y 471.943,Z 1180.166,A -85,B 0,C 180,E1 21896.014,E2 21896.014} C_VEL
LIN {X 0,Y 470.06,Z 1199.059,A -85,B 0,C 180,E1 21893.973,E2 21893.973} C_VEL
LIN {X 0,Y 468.445,Z 1216.434,A -85,B 0,C 180,E1 21891.797,E2 21891.797} C_VEL
LIN {X 0,Y 467.121,Z 1231.238,A -85,B 0,C 180,E1 21889.637,E2 21889.637} C_VEL
LIN {X 0,Y 466.029,Z 1244.568,A -85,B 0,C 180,E1 21887.353,E2 21887.353} C_VEL
LIN {X 0,Y 465.205,Z 1256.227,A -85,B 0,C 180,E1 21884.948,E2 21884.948} C_VEL
LIN {X 0,Y 464.642,Z 1265.782,A -85,B 0,C 180,E1 21882.555,E2 21882.555} C_VEL
LIN {X 0,Y 464.303,Z 1273.827,A -85,B 0,C 180,E1 21880.047,E2 21880.047} C_VEL
LIN {X 0,Y 464.144,Z 1279.873,A -85,B 0,C 180,E1 21877.553,E2 21877.553} C_VEL
LIN {X 0,Y 464.113,Z 1284.17,A -85,B 0,C 180,E1 21875.069,E2 21875.069} C_VEL
LIN {X 0,Y 464.103,Z 1286.811,A -85,B 0,C 180,E1 21872.595,E2 21872.595} C_VEL
LIN {X 0,Y 464.12,Z 1287.833,A -85,B 0,C 180,E1 21870.125,E2 21870.125} C_VEL
LIN {X 0,Y 464.087,Z 1287.2,A -85,B 0,C 180,E1 21867.532,E2 21867.532} C_VEL
LIN {X 0,Y 464.074,Z 1284.916,A -85,B 0,C 180,E1 21864.934,E2 21864.934} C_VEL
LIN {X 0,Y 464.093,Z 1280.914,A -85,B 0,C 180,E1 21862.325,E2 21862.325} C_VEL
LIN {X 0,Y 464.281,Z 1274.898,A -85,B 0,C 180,E1 21859.579,E2 21859.579} C_VEL
LIN {X 0,Y 464.681,Z 1267.318,A -85,B 0,C 180,E1 21856.944,E2 21856.944} C_VEL
LIN {X 0,Y 465.464,Z 1257.379,A -85,B 0,C 180,E1 21854.17,E2 21854.17} C_VEL
LIN {X 0,Y 466.635,Z 1245.781,A -85,B 0,C 180,E1 21851.513,E2 21851.513} C_VEL
LIN {X 0,Y 468.255,Z 1232.454,A -85,B 0,C 180,E1 21848.932,E2 21848.932} C_VEL
LIN {X 0,Y 470.45,Z 1216.575,A -85,B 0,C 180,E1 21846.318,E2 21846.318} C_VEL
LIN {X 0,Y 473.118,Z 1199.068,A -85,B 0,C 180,E1 21843.857,E2 21843.857} C_VEL
LIN {X 0,Y 476.075,Z 1180.844,A -85,B 0,C 180,E1 21841.645,E2 21841.645} C_VEL
LIN {X 0,Y 479.552,Z 1160.303,A -85,B 0,C 180,E1 21839.491,E2 21839.491} C_VEL
LIN {X 0,Y 483.582,Z 1137.01,A -85,B 0,C 180,E1 21837.412,E2 21837.412} C_VEL
LIN {X 0,Y 487.123,Z 1116.555,A -85,B 0,C 180,E1 21835.843,E2 21835.843} C_VEL
LIN {X 0,Y 491.258,Z 1092.515,A -85,B 0,C 180,E1 21834.26,E2 21834.26} C_VEL
LIN {X 0,Y 494.912,Z 1070.796,A -85,B 0,C 180,E1 21833.057,E2 21833.057} C_VEL
LIN {X 0,Y 499.058,Z 1044.767,A -85,B 0,C 180,E1 21831.862,E2 21831.862} C_VEL
LIN {X 0,Y 502.508,Z 1021.575,A -85,B 0,C 180,E1 21831.006,E2 21831.006} C_VEL
LIN {X 0,Y 505.741,Z 995.567,A -85,B 0,C 180,E1 21830.251,E2 21830.251} C_VEL
LIN {X 0,Y 507.83,Z 974.766,A -85,B 0,C 180,E1 21829.785,E2 21829.785} C_VEL
LIN {X 0,Y 510.878,Z 954.105,A -85,B 0,C 180,E1 21829.505,E2 21829.505} C_VEL
LIN {X 0,Y 513.027,Z 941.5,A -85,B 0,C 180,E1 21829.367,E2 21829.367} C_VEL
LIN {X 0,Y 509.956,Z 936.048,A -85,B 0,C 180,E1 21828.943,E2 21828.943} C_VEL
LIN {X 0,Y 503.723,Z 919.115,A -85,B 0,C 180,E1 21826.844,E2 21826.844} C_VEL
LIN {X 0,Y 499.747,Z 900.825,A -85,B 0,C 180,E1 21824.699,E2 21824.699} C_VEL
LIN {X 0,Y 498.15,Z 881.37,A -85,B 0,C 180,E1 21822.557,E2 21822.557} C_VEL
LIN {X 0,Y 498.982,Z 858.815,A -85,B 0,C 180,E1 21820.232,E2 21820.232} C_VEL
LIN {X 0,Y 505.12,Z 813.215,A -85,B 0,C 180,E1 21815.82,E2 21815.82} C_VEL
LIN {X 0,Y 510.082,Z 779.265,A -85,B 0,C 180,E1 21812.487,E2 21812.487} C_VEL
LIN {X 0,Y 514.92,Z 746.87,A -85,B 0,C 180,E1 21809.234,E2 21809.234} C_VEL
LIN {X 0,Y 515.687,Z 741.449,A -85,B 0,C 180,E1 21808.678,E2 21808.678} C_VEL
LIN {X 0,Y 508.098,Z 722.21,A -85,B 0,C 180,E1 21805.405,E2 21805.405} C_VEL
LIN {X 0,Y 500.788,Z 704.654,A -85,B 0,C 180,E1 21802.171,E2 21802.171} C_VEL
LIN {X 0,Y 493.915,Z 688.799,A -85,B 0,C 180,E1 21799.022,E2 21799.022} C_VEL
LIN {X 0,Y 486.74,Z 672.942,A -85,B 0,C 180,E1 21795.611,E2 21795.611} C_VEL
LIN {X 0,Y 480.397,Z 659.583,A -85,B 0,C 180,E1 21792.501,E2 21792.501} C_VEL
LIN {X 0,Y 474.796,Z 647.776,A -85,B 0,C 180,E1 21789.577,E2 21789.577} C_VEL
LIN {X 0,Y 470.125,Z 638.473,A -85,B 0,C 180,E1 21787.086,E2 21787.086} C_VEL
LIN {X 0,Y 467.991,Z 634.068,A -85,B 0,C 180,E1 21785.886,E2 21785.886} C_VEL
LIN {X 0,Y 466.313,Z 630.709,A -85,B 0,C 180,E1 21784.92,E2 21784.92} C_VEL
LIN {X 0,Y 466.17,Z 629.911,A -85,B 0,C 180,E1 21784.675,E2 21784.675} C_VEL
LIN {X 0,Y 466.163,Z 629.903,A -85,B 0,C 180,E1 21780.983,E2 21780.983} C_VEL
LIN {X 0,Y 466.169,Z 629.911,A -85,B 0,C 180,E1 21777.418,E2 21777.418} C_VEL
LIN {X 0,Y 466.169,Z 629.911,A -85,B 0,C 180,E1 21773.72,E2 21773.72} C_VEL
LIN {X 0,Y 466.17,Z 629.903,A -85,B 0,C 180,E1 21769.995,E2 21769.995} C_VEL
LIN {X 0,Y 466.18,Z 629.901,A -85,B 0,C 180,E1 21766.307,E2 21766.307} C_VEL
LIN {X 0,Y 466.17,Z 629.906,A -85,B 0,C 180,E1 21762.638,E2 21762.638} C_VEL
LIN {X 0,Y 466.168,Z 629.91,A -85,B 0,C 180,E1 21759.01,E2 21759.01} C_VEL
LIN {X 0,Y 466.178,Z 629.909,A -85,B 0,C 180,E1 21755.276,E2 21755.276} C_VEL
LIN {X 0,Y 466.18,Z 629.909,A -85,B 0,C 180,E1 21751.564,E2 21751.564} C_VEL
LIN {X 0,Y 466.166,Z 629.91,A -85,B 0,C 180,E1 21747.863,E2 21747.863} C_VEL
LIN {X 0,Y 466.168,Z 629.903,A -85,B 0,C 180,E1 21744.309,E2 21744.309} C_VEL
LIN {X 0,Y 466.183,Z 629.902,A -85,B 0,C 180,E1 21740.737,E2 21740.737} C_VEL
LIN {X 0,Y 466.164,Z 629.87,A -85,B 0,C 180,E1 21737.16,E2 21737.16} C_VEL
LIN {X 0,Y 466.177,Z 629.91,A -85,B 0,C 180,E1 21733.509,E2 21733.509} C_VEL
LIN {X 0,Y 466.202,Z 630.119,A -85,B 0,C 180,E1 21731.811,E2 21731.811} C_VEL
LIN {X 0,Y 475.723,Z 653.395,A -85,B 0,C 180,E1 21729.056,E2 21729.056} C_VEL
LIN {X 0,Y 483.189,Z 674.675,A -85,B 0,C 180,E1 21726.69,E2 21726.69} C_VEL
LIN {X 0,Y 487.6,Z 689.546,A -85,B 0,C 180,E1 21725.135,E2 21725.135} C_VEL
LIN {X 0,Y 484.868,Z 736.07,A -85,B 0,C 180,E1 21721.516,E2 21721.516} C_VEL
LIN {X 0,Y 482.068,Z 783.753,A -85,B 0,C 180,E1 21717.817,E2 21717.817} C_VEL
LIN {X 0,Y 479.66,Z 832.157,A -85,B 0,C 180,E1 21714.179,E2 21714.179} C_VEL
LIN {X 0,Y 478.856,Z 854.983,A -85,B 0,C 180,E1 21712.56,E2 21712.56} C_VEL
LIN {X 0,Y 479.479,Z 862.509,A -85,B 0,C 180,E1 21712.406,E2 21712.406} C_VEL
LIN {X 0,Y 476.635,Z 1023.308,A -85,B 0,C 180,E1 21709.958,E2 21709.958} C_VEL
LIN {X 0,Y 476.291,Z 1041.003,A -85,B 0,C 180,E1 21709.485,E2 21709.485} C_VEL
LIN {X 0,Y 475.635,Z 1057.515,A -85,B 0,C 180,E1 21708.824,E2 21708.824} C_VEL
LIN {X 0,Y 474.705,Z 1073.175,A -85,B 0,C 180,E1 21707.972,E2 21707.972} C_VEL
LIN {X 0,Y 473.512,Z 1088.805,A -85,B 0,C 180,E1 21706.877,E2 21706.877} C_VEL
LIN {X 0,Y 472.2,Z 1103.321,A -85,B 0,C 180,E1 21705.598,E2 21705.598} C_VEL
LIN {X 0,Y 470.817,Z 1116.611,A -85,B 0,C 180,E1 21704.134,E2 21704.134} C_VEL
LIN {X 0,Y 469.501,Z 1128.326,A -85,B 0,C 180,E1 21702.544,E2 21702.544} C_VEL
LIN {X 0,Y 468.308,Z 1138.597,A -85,B 0,C 180,E1 21700.828,E2 21700.828} C_VEL
LIN {X 0,Y 467.283,Z 1147.45,A -85,B 0,C 180,E1 21698.985,E2 21698.985} C_VEL
LIN {X 0,Y 466.459,Z 1154.785,A -85,B 0,C 180,E1 21697.016,E2 21697.016} C_VEL
LIN {X 0,Y 466.207,Z 1157.206,A -85,B 0,C 180,E1 21696.233,E2 21696.233} C_VEL
LIN {X 0,Y 464.971,Z 1159.765,A -85,B 0,C 180,E1 21695.34,E2 21695.34} C_VEL
LIN {X 0,Y 459.841,Z 1164.155,A -85,B 0,C 180,E1 21693.587,E2 21693.587} C_VEL
LIN {X 0,Y 457.637,Z 1166.125,A -85,B 0,C 180,E1 21692.464,E2 21692.464} C_VEL
LIN {X 0,Y 457.458,Z 1166.55,A -85,B 0,C 180,E1 21692.121,E2 21692.121} C_VEL
LIN {X 0,Y 457.321,Z 1168.318,A -85,B 0,C 180,E1 21689.873,E2 21689.873} C_VEL
LIN {X 0,Y 457.344,Z 1168.226,A -85,B 0,C 180,E1 21687.618,E2 21687.618} C_VEL
LIN {X 0,Y 457.546,Z 1166.333,A -85,B 0,C 180,E1 21685.361,E2 21685.361} C_VEL
LIN {X 0,Y 457.973,Z 1162.592,A -85,B 0,C 180,E1 21683.102,E2 21683.102} C_VEL
LIN {X 0,Y 458.613,Z 1157.135,A -85,B 0,C 180,E1 21680.967,E2 21680.967} C_VEL
LIN {X 0,Y 459.551,Z 1149.677,A -85,B 0,C 180,E1 21678.833,E2 21678.833} C_VEL
LIN {X 0,Y 460.662,Z 1141.178,A -85,B 0,C 180,E1 21676.952,E2 21676.952} C_VEL
LIN {X 0,Y 461.951,Z 1131.252,A -85,B 0,C 180,E1 21675.201,E2 21675.201} C_VEL
LIN {X 0,Y 463.364,Z 1119.876,A -85,B 0,C 180,E1 21673.578,E2 21673.578} C_VEL
LIN {X 0,Y 464.909,Z 1106.419,A -85,B 0,C 180,E1 21672.022,E2 21672.022} C_VEL
LIN {X 0,Y 466.341,Z 1092.45,A -85,B 0,C 180,E1 21670.718,E2 21670.718} C_VEL
LIN {X 0,Y 467.625,Z 1077.376,A -85,B 0,C 180,E1 21669.601,E2 21669.601} C_VEL
LIN {X 0,Y 468.704,Z 1061.231,A -85,B 0,C 180,E1 21668.669,E2 21668.669} C_VEL
LIN {X 0,Y 469.509,Z 1044.172,A -85,B 0,C 180,E1 21667.936,E2 21667.936} C_VEL
LIN {X 0,Y 469.936,Z 1026.776,A -85,B 0,C 180,E1 21667.433,E2 21667.433} C_VEL
LIN {X 0,Y 470.613,Z 979.745,A -85,B 0,C 180,E1 21666.669,E2 21666.669} C_VEL
LIN {X 0,Y 472.876,Z 860.245,A -85,B 0,C 180,E1 21664.833,E2 21664.833} C_VEL
LIN {X 0,Y 472.288,Z 854.941,A -85,B 0,C 180,E1 21664.68,E2 21664.68} C_VEL
LIN {X 0,Y 474.393,Z 809.981,A -85,B 0,C 180,E1 21661.345,E2 21661.345} C_VEL
LIN {X 0,Y 477.217,Z 762.985,A -85,B 0,C 180,E1 21657.703,E2 21657.703} C_VEL
LIN {X 0,Y 480.127,Z 717.252,A -85,B 0,C 180,E1 21654.107,E2 21654.107} C_VEL
LIN {X 0,Y 481.55,Z 693.391,A -85,B 0,C 180,E1 21652.225,E2 21652.225} C_VEL
LIN {X 0,Y 474.966,Z 672.56,A -85,B 0,C 180,E1 21649.928,E2 21649.928} C_VEL
LIN {X 0,Y 467.23,Z 651.964,A -85,B 0,C 180,E1 21647.499,E2 21647.499} C_VEL
LIN {X 0,Y 468.515,Z 652.322,A -85,B 0,C 180,E1 21647.236,E2 21647.236} C_VEL
LIN {X 0,Y 471.061,Z 657.346,A -85,B 0,C 180,E1 21646.275,E2 21646.275} C_VEL
LIN {X 0,Y 488.899,Z 682.289,A -85,B 0,C 180,E1 21643.507,E2 21643.507} C_VEL
LIN {X 0,Y 506.854,Z 708.57,A -85,B 0,C 180,E1 21640.989,E2 21640.989} C_VEL
LIN {X 0,Y 508.728,Z 711.684,A -85,B 0,C 180,E1 21640.729,E2 21640.729} C_VEL
LIN {X 0,Y 492.4,Z 974.784,A -85,B 0,C 180,E1 21635.616,E2 21635.616} C_VEL
LIN {X 0,Y 490.747,Z 997.919,A -85,B 0,C 180,E1 21634.947,E2 21634.947} C_VEL
LIN {X 0,Y 488.583,Z 1020.892,A -85,B 0,C 180,E1 21634.072,E2 21634.072} C_VEL
LIN {X 0,Y 486.08,Z 1042.582,A -85,B 0,C 180,E1 21633.033,E2 21633.033} C_VEL
LIN {X 0,Y 483.164,Z 1063.82,A -85,B 0,C 180,E1 21631.782,E2 21631.782} C_VEL
LIN {X 0,Y 479.93,Z 1085.068,A -85,B 0,C 180,E1 21630.277,E2 21630.277} C_VEL
LIN {X 0,Y 476.798,Z 1103.961,A -85,B 0,C 180,E1 21628.701,E2 21628.701} C_VEL
LIN {X 0,Y 473.443,Z 1122.489,A -85,B 0,C 180,E1 21626.87,E2 21626.87} C_VEL
LIN {X 0,Y 470.174,Z 1140.074,A -85,B 0,C 180,E1 21624.835,E2 21624.835} C_VEL
LIN {X 0,Y 467.206,Z 1155.836,A -85,B 0,C 180,E1 21622.718,E2 21622.718} C_VEL
LIN {X 0,Y 464.462,Z 1170.404,A -85,B 0,C 180,E1 21620.411,E2 21620.411} C_VEL
LIN {X 0,Y 462.002,Z 1183.948,A -85,B 0,C 180,E1 21617.898,E2 21617.898} C_VEL
LIN {X 0,Y 460.085,Z 1195.515,A -85,B 0,C 180,E1 21615.375,E2 21615.375} C_VEL
LIN {X 0,Y 458.616,Z 1205.135,A -85,B 0,C 180,E1 21612.849,E2 21612.849} C_VEL
LIN {X 0,Y 457.451,Z 1214.26,A -85,B 0,C 180,E1 21609.944,E2 21609.944} C_VEL
LIN {X 0,Y 456.764,Z 1221.214,A -85,B 0,C 180,E1 21607.168,E2 21607.168} C_VEL
LIN {X 0,Y 456.369,Z 1226.359,A -85,B 0,C 180,E1 21604.398,E2 21604.398} C_VEL
LIN {X 0,Y 456.194,Z 1230.144,A -85,B 0,C 180,E1 21601.507,E2 21601.507} C_VEL
LIN {X 0,Y 456.145,Z 1232.047,A -85,B 0,C 180,E1 21598.995,E2 21598.995} C_VEL
LIN {X 0,Y 456.158,Z 1232.725,A -85,B 0,C 180,E1 21596.104,E2 21596.104} C_VEL
LIN {X 0,Y 456.212,Z 1231.932,A -85,B 0,C 180,E1 21593.456,E2 21593.456} C_VEL
LIN {X 0,Y 456.392,Z 1229.556,A -85,B 0,C 180,E1 21590.67,E2 21590.67} C_VEL
LIN {X 0,Y 456.765,Z 1225.716,A -85,B 0,C 180,E1 21587.869,E2 21587.869} C_VEL
LIN {X 0,Y 457.401,Z 1220.444,A -85,B 0,C 180,E1 21585.181,E2 21585.181} C_VEL
LIN {X 0,Y 458.481,Z 1213.26,A -85,B 0,C 180,E1 21582.353,E2 21582.353} C_VEL
LIN {X 0,Y 460.018,Z 1204.703,A -85,B 0,C 180,E1 21579.649,E2 21579.649} C_VEL
LIN {X 0,Y 461.973,Z 1194.679,A -85,B 0,C 180,E1 21577.071,E2 21577.071} C_VEL
LIN {X 0,Y 464.356,Z 1183.342,A -85,B 0,C 180,E1 21574.627,E2 21574.627} C_VEL
LIN {X 0,Y 467.097,Z 1170.775,A -85,B 0,C 180,E1 21572.321,E2 21572.321} C_VEL
LIN {X 0,Y 470.324,Z 1155.914,A -85,B 0,C 180,E1 21570.026,E2 21570.026} C_VEL
LIN {X 0,Y 473.469,Z 1140.868,A -85,B 0,C 180,E1 21568.061,E2 21568.061} C_VEL
LIN {X 0,Y 476.884,Z 1123.817,A -85,B 0,C 180,E1 21566.166,E2 21566.166} C_VEL
LIN {X 0,Y 479.938,Z 1107.384,A -85,B 0,C 180,E1 21564.607,E2 21564.607} C_VEL
LIN {X 0,Y 483.025,Z 1088.46,A -85,B 0,C 180,E1 21563.107,E2 21563.107} C_VEL
LIN {X 0,Y 485.659,Z 1069.435,A -85,B 0,C 180,E1 21561.855,E2 21561.855} C_VEL
LIN {X 0,Y 487.959,Z 1049.24,A -85,B 0,C 180,E1 21560.768,E2 21560.768} C_VEL
LIN {X 0,Y 489.739,Z 1028.914,A -85,B 0,C 180,E1 21559.898,E2 21559.898} C_VEL
LIN {X 0,Y 490.954,Z 1007.742,A -85,B 0,C 180,E1 21559.206,E2 21559.206} C_VEL
LIN {X 0,Y 492.966,Z 968.452,A -85,B 0,C 180,E1 21558.28,E2 21558.28} C_VEL
LIN {X 0,Y 497.547,Z 923.115,A -85,B 0,C 180,E1 21557.234,E2 21557.234} C_VEL
LIN {X 0,Y 503.864,Z 879.366,A -85,B 0,C 180,E1 21556.121,E2 21556.121} C_VEL
LIN {X 0,Y 506.872,Z 861.966,A -85,B 0,C 180,E1 21555.65,E2 21555.65} C_VEL
LIN {X 0,Y 502.729,Z 873.626,A -85,B 0,C 180,E1 21554.456,E2 21554.456} C_VEL
LIN {X 0,Y 500.697,Z 885.389,A -85,B 0,C 180,E1 21553.205,E2 21553.205} C_VEL
LIN {X 0,Y 500.84,Z 898.258,A -85,B 0,C 180,E1 21551.85,E2 21551.85} C_VEL
LIN {X 0,Y 503.124,Z 911.924,A -85,B 0,C 180,E1 21550.497,E2 21550.497} C_VEL
LIN {X 0,Y 505.348,Z 920.037,A -85,B 0,C 180,E1 21549.729,E2 21549.729} C_VEL
LIN {X 0,Y 499.156,Z 940.917,A -85,B 0,C 180,E1 21549.64,E2 21549.64} C_VEL
LIN {X 0,Y 494.467,Z 959.321,A -85,B 0,C 180,E1 21549.353,E2 21549.353} C_VEL
LIN {X 0,Y 490.715,Z 977.506,A -85,B 0,C 180,E1 21548.864,E2 21548.864} C_VEL
LIN {X 0,Y 485.288,Z 1012.533,A -85,B 0,C 180,E1 21547.509,E2 21547.509} C_VEL
LIN {X 0,Y 480.299,Z 1046.467,A -85,B 0,C 180,E1 21545.951,E2 21545.951} C_VEL
LIN {X 0,Y 475.902,Z 1079.065,A -85,B 0,C 180,E1 21544.177,E2 21544.177} C_VEL
LIN {X 0,Y 472.17,Z 1109.281,A -85,B 0,C 180,E1 21542.254,E2 21542.254} C_VEL
LIN {X 0,Y 468.789,Z 1138.681,A -85,B 0,C 180,E1 21540.083,E2 21540.083} C_VEL
LIN {X 0,Y 466.143,Z 1162.787,A -85,B 0,C 180,E1 21538.02,E2 21538.02} C_VEL
LIN {X 0,Y 463.772,Z 1185.104,A -85,B 0,C 180,E1 21535.819,E2 21535.819} C_VEL
LIN {X 0,Y 461.866,Z 1203.767,A -85,B 0,C 180,E1 21533.687,E2 21533.687} C_VEL
LIN {X 0,Y 460.187,Z 1220.84,A -85,B 0,C 180,E1 21531.411,E2 21531.411} C_VEL
LIN {X 0,Y 458.835,Z 1235.742,A -85,B 0,C 180,E1 21529.081,E2 21529.081} C_VEL
LIN {X 0,Y 457.792,Z 1248.319,A -85,B 0,C 180,E1 21526.758,E2 21526.758} C_VEL
LIN {X 0,Y 457.05,Z 1258.76,A -85,B 0,C 180,E1 21524.443,E2 21524.443} C_VEL
LIN {X 0,Y 456.56,Z 1267.764,A -85,B 0,C 180,E1 21522.01,E2 21522.01} C_VEL
LIN {X 0,Y 456.25,Z 1275.24,A -85,B 0,C 180,E1 21519.462,E2 21519.462} C_VEL
LIN {X 0,Y 456.133,Z 1280.844,A -85,B 0,C 180,E1 21516.926,E2 21516.926} C_VEL
LIN {X 0,Y 456.11,Z 1284.624,A -85,B 0,C 180,E1 21514.402,E2 21514.402} C_VEL
LIN {X 0,Y 456.128,Z 1286.77,A -85,B 0,C 180,E1 21511.886,E2 21511.886} C_VEL
LIN {X 0,Y 456.121,Z 1287.322,A -85,B 0,C 180,E1 21509.374,E2 21509.374} C_VEL
LIN {X 0,Y 456.101,Z 1286.281,A -85,B 0,C 180,E1 21506.86,E2 21506.86} C_VEL
LIN {X 0,Y 456.079,Z 1283.506,A -85,B 0,C 180,E1 21504.214,E2 21504.214} C_VEL
LIN {X 0,Y 456.143,Z 1279.06,A -85,B 0,C 180,E1 21501.556,E2 21501.556} C_VEL
LIN {X 0,Y 456.362,Z 1272.832,A -85,B 0,C 180,E1 21498.885,E2 21498.885} C_VEL
LIN {X 0,Y 456.886,Z 1264.392,A -85,B 0,C 180,E1 21496.072,E2 21496.072} C_VEL
LIN {X 0,Y 457.754,Z 1254.323,A -85,B 0,C 180,E1 21493.375,E2 21493.375} C_VEL
LIN {X 0,Y 459.102,Z 1242.229,A -85,B 0,C 180,E1 21490.67,E2 21490.67} C_VEL
LIN {X 0,Y 461.076,Z 1227.092,A -85,B 0,C 180,E1 21487.833,E2 21487.833} C_VEL
LIN {X 0,Y 463.61,Z 1209.995,A -85,B 0,C 180,E1 21485.132,E2 21485.132} C_VEL
LIN {X 0,Y 466.512,Z 1191.998,A -85,B 0,C 180,E1 21482.701,E2 21482.701} C_VEL
LIN {X 0,Y 469.76,Z 1172.966,A -85,B 0,C 180,E1 21480.481,E2 21480.481} C_VEL
LIN {X 0,Y 473.525,Z 1151.726,A -85,B 0,C 180,E1 21478.345,E2 21478.345} C_VEL
LIN {X 0,Y 477.196,Z 1131.06,A -85,B 0,C 180,E1 21476.562,E2 21476.562} C_VEL
LIN {X 0,Y 481.294,Z 1108.491,A -85,B 0,C 180,E1 21474.87,E2 21474.87} C_VEL
LIN {X 0,Y 485.23,Z 1086.098,A -85,B 0,C 180,E1 21473.452,E2 21473.452} C_VEL
LIN {X 0,Y 489.278,Z 1062.664,A -85,B 0,C 180,E1 21472.19,E2 21472.19} C_VEL
LIN {X 0,Y 493.066,Z 1039.172,A -85,B 0,C 180,E1 21471.157,E2 21471.157} C_VEL
LIN {X 0,Y 497.014,Z 1012.918,A -85,B 0,C 180,E1 21470.23,E2 21470.23} C_VEL
LIN {X 0,Y 499.917,Z 988.427,A -85,B 0,C 180,E1 21469.547,E2 21469.547} C_VEL
LIN {X 0,Y 502.274,Z 967.785,A -85,B 0,C 180,E1 21469.133,E2 21469.133} C_VEL
LIN {X 0,Y 506.096,Z 944.122,A -85,B 0,C 180,E1 21468.851,E2 21468.851} C_VEL
LIN {X 0,Y 500.291,Z 933.402,A -85,B 0,C 180,E1 21468.03,E2 21468.03} C_VEL
LIN {X 0,Y 494.947,Z 916.107,A -85,B 0,C 180,E1 21465.905,E2 21465.905} C_VEL
LIN {X 0,Y 491.921,Z 898.168,A -85,B 0,C 180,E1 21463.818,E2 21463.818} C_VEL
LIN {X 0,Y 491.062,Z 877.785,A -85,B 0,C 180,E1 21461.59,E2 21461.59} C_VEL
LIN {X 0,Y 492.644,Z 854.976,A -85,B 0,C 180,E1 21459.261,E2 21459.261} C_VEL
LIN {X 0,Y 498.298,Z 815.862,A -85,B 0,C 180,E1 21455.444,E2 21455.444} C_VEL
LIN {X 0,Y 503.524,Z 781.254,A -85,B 0,C 180,E1 21452.017,E2 21452.017} C_VEL
LIN {X 0,Y 508.527,Z 748.77,A -85,B 0,C 180,E1 21448.729,E2 21448.729} C_VEL
LIN {X 0,Y 509.046,Z 745.261,A -85,B 0,C 180,E1 21448.365,E2 21448.365} C_VEL
LIN {X 0,Y 501.66,Z 726.437,A -85,B 0,C 180,E1 21445.122,E2 21445.122} C_VEL
LIN {X 0,Y 494.151,Z 708.283,A -85,B 0,C 180,E1 21441.734,E2 21441.734} C_VEL
LIN {X 0,Y 486.56,Z 690.775,A -85,B 0,C 180,E1 21438.202,E2 21438.202} C_VEL
LIN {X 0,Y 480.067,Z 676.637,A -85,B 0,C 180,E1 21435.091,E2 21435.091} C_VEL
LIN {X 0,Y 474.491,Z 664.714,A -85,B 0,C 180,E1 21432.289,E2 21432.289} C_VEL
LIN {X 0,Y 469.129,Z 653.331,A -85,B 0,C 180,E1 21429.446,E2 21429.446} C_VEL
LIN {X 0,Y 464.449,Z 643.985,A -85,B 0,C 180,E1 21426.924,E2 21426.924} C_VEL
LIN {X 0,Y 462.062,Z 639.243,A -85,B 0,C 180,E1 21425.588,E2 21425.588} C_VEL
LIN {X 0,Y 459.959,Z 634.958,A -85,B 0,C 180,E1 21424.364,E2 21424.364} C_VEL
LIN {X 0,Y 458.33,Z 631.527,A -85,B 0,C 180,E1 21423.377,E2 21423.377} C_VEL
LIN {X 0,Y 458.223,Z 630.893,A -85,B 0,C 180,E1 21423.19,E2 21423.19} C_VEL
LIN {X 0,Y 458.241,Z 630.9,A -85,B 0,C 180,E1 21419.5,E2 21419.5} C_VEL
LIN {X 0,Y 458.235,Z 630.891,A -85,B 0,C 180,E1 21415.673,E2 21415.673} C_VEL
LIN {X 0,Y 458.231,Z 630.896,A -85,B 0,C 180,E1 21411.972,E2 21411.972} C_VEL
LIN {X 0,Y 458.229,Z 630.903,A -85,B 0,C 180,E1 21408.291,E2 21408.291} C_VEL
LIN {X 0,Y 458.236,Z 630.901,A -85,B 0,C 180,E1 21404.561,E2 21404.561} C_VEL
LIN {X 0,Y 458.24,Z 630.896,A -85,B 0,C 180,E1 21400.762,E2 21400.762} C_VEL
LIN {X 0,Y 458.225,Z 630.894,A -85,B 0,C 180,E1 21397.043,E2 21397.043} C_VEL
LIN {X 0,Y 458.235,Z 630.891,A -85,B 0,C 180,E1 21393.428,E2 21393.428} C_VEL
LIN {X 0,Y 458.228,Z 630.893,A -85,B 0,C 180,E1 21389.731,E2 21389.731} C_VEL
LIN {X 0,Y 458.24,Z 630.893,A -85,B 0,C 180,E1 21386.009,E2 21386.009} C_VEL
LIN {X 0,Y 458.243,Z 630.893,A -85,B 0,C 180,E1 21382.171,E2 21382.171} C_VEL
LIN {X 0,Y 458.226,Z 630.884,A -85,B 0,C 180,E1 21378.443,E2 21378.443} C_VEL
LIN {X 0,Y 458.238,Z 630.885,A -85,B 0,C 180,E1 21374.634,E2 21374.634} C_VEL
LIN {X 0,Y 458.248,Z 631.003,A -85,B 0,C 180,E1 21372.501,E2 21372.501} C_VEL
LIN {X 0,Y 459.529,Z 634.354,A -85,B 0,C 180,E1 21372.099,E2 21372.099} C_VEL
LIN {X 0,Y 467.372,Z 653.027,A -85,B 0,C 180,E1 21369.821,E2 21369.821} C_VEL
LIN {X 0,Y 474.463,Z 672.428,A -85,B 0,C 180,E1 21367.59,E2 21367.59} C_VEL
LIN {X 0,Y 480.515,Z 692.014,A -85,B 0,C 180,E1 21365.488,E2 21365.488} C_VEL
LIN {X 0,Y 477.748,Z 737.778,A -85,B 0,C 180,E1 21361.899,E2 21361.899} C_VEL
LIN {X 0,Y 474.873,Z 785.054,A -85,B 0,C 180,E1 21358.208,E2 21358.208} C_VEL
LIN {X 0,Y 472.349,Z 833.904,A -85,B 0,C 180,E1 21354.511,E2 21354.511} C_VEL
LIN {X 0,Y 471.546,Z 855.975,A -85,B 0,C 180,E1 21352.938,E2 21352.938} C_VEL
LIN {X 0,Y 472.144,Z 863.417,A -85,B 0,C 180,E1 21352.784,E2 21352.784} C_VEL
LIN {X 0,Y 469.189,Z 1023.975,A -85,B 0,C 180,E1 21350.304,E2 21350.304} C_VEL
LIN {X 0,Y 468.831,Z 1041.773,A -85,B 0,C 180,E1 21349.824,E2 21349.824} C_VEL
LIN {X 0,Y 468.134,Z 1058.652,A -85,B 0,C 180,E1 21349.137,E2 21349.137} C_VEL
LIN {X 0,Y 467.168,Z 1074.275,A -85,B 0,C 180,E1 21348.272,E2 21348.272} C_VEL
LIN {X 0,Y 465.93,Z 1089.878,A -85,B 0,C 180,E1 21347.16,E2 21347.16} C_VEL
LIN {X 0,Y 464.566,Z 1104.373,A -85,B 0,C 180,E1 21345.861,E2 21345.861} C_VEL
LIN {X 0,Y 463.128,Z 1117.642,A -85,B 0,C 180,E1 21344.374,E2 21344.374} C_VEL
LIN {X 0,Y 461.757,Z 1129.345,A -85,B 0,C 180,E1 21342.758,E2 21342.758} C_VEL
LIN {X 0,Y 460.513,Z 1139.604,A -85,B 0,C 180,E1 21341.013,E2 21341.013} C_VEL
LIN {X 0,Y 459.441,Z 1148.446,A -85,B 0,C 180,E1 21339.14,E2 21339.14} C_VEL
LIN {X 0,Y 458.577,Z 1155.771,A -85,B 0,C 180,E1 21337.138,E2 21337.138} C_VEL
LIN {X 0,Y 457.945,Z 1161.577,A -85,B 0,C 180,E1 21335.009,E2 21335.009} C_VEL
LIN {X 0,Y 457.554,Z 1165.567,A -85,B 0,C 180,E1 21332.879,E2 21332.879} C_VEL
LIN {X 0,Y 457.458,Z 1166.55,A -85,B 0,C 180,E1 21332.121,E2 21332.121} C_VEL
LIN {X 0,Y 456.393,Z 1167.688,A -85,B 0,C 180,E1 21331.166,E2 21331.166} C_VEL
LIN {X 0,Y 451.91,Z 1169.191,A -85,B 0,C 180,E1 21329.428,E2 21329.428} C_VEL
LIN {X 0,Y 449.658,Z 1169.417,A -85,B 0,C 180,E1 21328.254,E2 21328.254} C_VEL
LIN {X 0,Y 449.398,Z 1169.264,A -85,B 0,C 180,E1 21327.759,E2 21327.759} C_VEL
LIN {X 0,Y 449.585,Z 1167.578,A -85,B 0,C 180,E1 21325.534,E2 21325.534} C_VEL
LIN {X 0,Y 450.005,Z 1164.012,A -85,B 0,C 180,E1 21323.235,E2 21323.235} C_VEL
LIN {X 0,Y 450.659,Z 1158.824,A -85,B 0,C 180,E1 21321.064,E2 21321.064} C_VEL
LIN {X 0,Y 451.542,Z 1152.072,A -85,B 0,C 180,E1 21319.02,E2 21319.02} C_VEL
LIN {X 0,Y 452.73,Z 1143.302,A -85,B 0,C 180,E1 21316.979,E2 21316.979} C_VEL
LIN {X 0,Y 454.063,Z 1133.556,A -85,B 0,C 180,E1 21315.178,E2 21315.178} C_VEL
LIN {X 0,Y 455.498,Z 1122.691,A -85,B 0,C 180,E1 21313.549,E2 21313.549} C_VEL
LIN {X 0,Y 457.071,Z 1109.615,A -85,B 0,C 180,E1 21311.967,E2 21311.967} C_VEL
LIN {X 0,Y 458.61,Z 1095.407,A -85,B 0,C 180,E1 21310.579,E2 21310.579} C_VEL
LIN {X 0,Y 459.945,Z 1080.957,A -85,B 0,C 180,E1 21309.445,E2 21309.445} C_VEL
LIN {X 0,Y 461.092,Z 1065.312,A -85,B 0,C 180,E1 21308.482,E2 21308.482} C_VEL
LIN {X 0,Y 461.977,Z 1048.293,A -85,B 0,C 180,E1 21307.699,E2 21307.699} C_VEL
LIN {X 0,Y 462.51,Z 1030.796,A -85,B 0,C 180,E1 21307.14,E2 21307.14} C_VEL
LIN {X 0,Y 462.736,Z 1007.431,A -85,B 0,C 180,E1 21306.706,E2 21306.706} C_VEL
LIN {X 0,Y 465.628,Z 861.117,A -85,B 0,C 180,E1 21304.425,E2 21304.425} C_VEL
LIN {X 0,Y 465.048,Z 855.92,A -85,B 0,C 180,E1 21304.275,E2 21304.275} C_VEL
LIN {X 0,Y 467.242,Z 811.266,A -85,B 0,C 180,E1 21300.935,E2 21300.935} C_VEL
LIN {X 0,Y 470.075,Z 765.793,A -85,B 0,C 180,E1 21297.387,E2 21297.387} C_VEL
LIN {X 0,Y 473.137,Z 719.46,A -85,B 0,C 180,E1 21293.719,E2 21293.719} C_VEL
LIN {X 0,Y 474.518,Z 696.16,A -85,B 0,C 180,E1 21291.872,E2 21291.872} C_VEL
LIN {X 0,Y 468.31,Z 676.434,A -85,B 0,C 180,E1 21289.662,E2 21289.662} C_VEL
LIN {X 0,Y 461.738,Z 658.539,A -85,B 0,C 180,E1 21287.495,E2 21287.495} C_VEL
LIN {X 0,Y 463.487,Z 659.154,A -85,B 0,C 180,E1 21287.147,E2 21287.147} C_VEL
LIN {X 0,Y 481.03,Z 683.437,A -85,B 0,C 180,E1 21284.351,E2 21284.351} C_VEL
LIN {X 0,Y 499.126,Z 709.944,A -85,B 0,C 180,E1 21281.713,E2 21281.713} C_VEL
LIN {X 0,Y 502.397,Z 715.193,A -85,B 0,C 180,E1 21281.253,E2 21281.253} C_VEL
LIN {X 0,Y 485.514,Z 975.554,A -85,B 0,C 180,E1 21276.086,E2 21276.086} C_VEL
LIN {X 0,Y 483.819,Z 998.561,A -85,B 0,C 180,E1 21275.411,E2 21275.411} C_VEL
LIN {X 0,Y 481.676,Z 1020.845,A -85,B 0,C 180,E1 21274.557,E2 21274.557} C_VEL
LIN {X 0,Y 479.147,Z 1042.167,A -85,B 0,C 180,E1 21273.526,E2 21273.526} C_VEL
LIN {X 0,Y 476.233,Z 1062.979,A -85,B 0,C 180,E1 21272.3,E2 21272.3} C_VEL
LIN {X 0,Y 473.024,Z 1083.728,A -85,B 0,C 180,E1 21270.838,E2 21270.838} C_VEL
LIN {X 0,Y 469.708,Z 1103.086,A -85,B 0,C 180,E1 21269.214,E2 21269.214} C_VEL
LIN {X 0,Y 466.356,Z 1121.263,A -85,B 0,C 180,E1 21267.42,E2 21267.42} C_VEL
LIN {X 0,Y 463.079,Z 1138.461,A -85,B 0,C 180,E1 21265.448,E2 21265.448} C_VEL
LIN {X 0,Y 459.973,Z 1154.41,A -85,B 0,C 180,E1 21263.306,E2 21263.306} C_VEL
LIN {X 0,Y 457.133,Z 1168.963,A -85,B 0,C 180,E1 21261.022,E2 21261.022} C_VEL
LIN {X 0,Y 454.631,Z 1182.38,A -85,B 0,C 180,E1 21258.57,E2 21258.57} C_VEL
LIN {X 0,Y 452.561,Z 1194.073,A -85,B 0,C 180,E1 21256.032,E2 21256.032} C_VEL
LIN {X 0,Y 450.895,Z 1204.515,A -85,B 0,C 180,E1 21253.334,E2 21253.334} C_VEL
LIN {X 0,Y 449.716,Z 1213.222,A -85,B 0,C 180,E1 21250.634,E2 21250.634} C_VEL
LIN {X 0,Y 448.94,Z 1220.108,A -85,B 0,C 180,E1 21247.937,E2 21247.937} C_VEL
LIN {X 0,Y 448.452,Z 1225.972,A -85,B 0,C 180,E1 21244.989,E2 21244.989} C_VEL
LIN {X 0,Y 448.242,Z 1229.787,A -85,B 0,C 180,E1 21242.301,E2 21242.301} C_VEL
LIN {X 0,Y 448.166,Z 1232.251,A -85,B 0,C 180,E1 21239.489,E2 21239.489} C_VEL
LIN {X 0,Y 448.161,Z 1233.222,A -85,B 0,C 180,E1 21236.931,E2 21236.931} C_VEL
LIN {X 0,Y 448.224,Z 1232.808,A -85,B 0,C 180,E1 21234.11,E2 21234.11} C_VEL
LIN {X 0,Y 448.369,Z 1230.976,A -85,B 0,C 180,E1 21231.278,E2 21231.278} C_VEL
LIN {X 0,Y 448.683,Z 1227.664,A -85,B 0,C 180,E1 21228.56,E2 21228.56} C_VEL
LIN {X 0,Y 449.35,Z 1222.44,A -85,B 0,C 180,E1 21225.568,E2 21225.568} C_VEL
LIN {X 0,Y 450.423,Z 1215.762,A -85,B 0,C 180,E1 21222.694,E2 21222.694} C_VEL
LIN {X 0,Y 451.929,Z 1207.547,A -85,B 0,C 180,E1 21219.944,E2 21219.944} C_VEL
LIN {X 0,Y 454.004,Z 1197.517,A -85,B 0,C 180,E1 21217.193,E2 21217.193} C_VEL
LIN {X 0,Y 456.441,Z 1186.702,A -85,B 0,C 180,E1 21214.712,E2 21214.712} C_VEL
LIN {X 0,Y 459.395,Z 1173.813,A -85,B 0,C 180,E1 21212.239,E2 21212.239} C_VEL
LIN {X 0,Y 462.525,Z 1160.248,A -85,B 0,C 180,E1 21210.041,E2 21210.041} C_VEL
LIN {X 0,Y 465.929,Z 1145.243,A -85,B 0,C 180,E1 21207.961,E2 21207.961} C_VEL
LIN {X 0,Y 469.389,Z 1129.24,A -85,B 0,C 180,E1 21206.074,E2 21206.074} C_VEL
LIN {X 0,Y 472.804,Z 1112,A -85,B 0,C 180,E1 21204.364,E2 21204.364} C_VEL
LIN {X 0,Y 476.034,Z 1093.95,A -85,B 0,C 180,E1 21202.851,E2 21202.851} C_VEL
LIN {X 0,Y 478.986,Z 1074.951,A -85,B 0,C 180,E1 21201.521,E2 21201.521} C_VEL
LIN {X 0,Y 481.388,Z 1056.73,A -85,B 0,C 180,E1 21200.459,E2 21200.459} C_VEL
LIN {X 0,Y 483.556,Z 1035.589,A -85,B 0,C 180,E1 21199.473,E2 21199.473} C_VEL
LIN {X 0,Y 485.139,Z 1013.341,A -85,B 0,C 180,E1 21198.677,E2 21198.677} C_VEL
LIN {X 0,Y 487.346,Z 976.685,A -85,B 0,C 180,E1 21197.734,E2 21197.734} C_VEL
LIN {X 0,Y 491.932,Z 936.694,A -85,B 0,C 180,E1 21196.751,E2 21196.751} C_VEL
LIN {X 0,Y 498.521,Z 896.507,A -85,B 0,C 180,E1 21195.689,E2 21195.689} C_VEL
LIN {X 0,Y 502.11,Z 878.439,A -85,B 0,C 180,E1 21195.186,E2 21195.186} C_VEL
LIN {X 0,Y 498.732,Z 889.851,A -85,B 0,C 180,E1 21193.942,E2 21193.942} C_VEL
LIN {X 0,Y 497.56,Z 901.643,A -85,B 0,C 180,E1 21192.629,E2 21192.629} C_VEL
LIN {X 0,Y 498.517,Z 914.596,A -85,B 0,C 180,E1 21191.271,E2 21191.271} C_VEL
LIN {X 0,Y 500.049,Z 922.315,A -85,B 0,C 180,E1 21190.489,E2 21190.489} C_VEL
LIN {X 0,Y 494.19,Z 942.333,A -85,B 0,C 180,E1 21190.386,E2 21190.386} C_VEL
LIN {X 0,Y 489.236,Z 961.411,A -85,B 0,C 180,E1 21190.057,E2 21190.057} C_VEL
LIN {X 0,Y 485.346,Z 979.344,A -85,B 0,C 180,E1 21189.539,E2 21189.539} C_VEL
LIN {X 0,Y 479.17,Z 1015.306,A -85,B 0,C 180,E1 21188.071,E2 21188.071} C_VEL
LIN {X 0,Y 473.765,Z 1048.717,A -85,B 0,C 180,E1 21186.458,E2 21186.458} C_VEL
LIN {X 0,Y 469.005,Z 1081.049,A -85,B 0,C 180,E1 21184.621,E2 21184.621} C_VEL
LIN {X 0,Y 464.815,Z 1112.529,A -85,B 0,C 180,E1 21182.535,E2 21182.535} C_VEL
LIN {X 0,Y 461.454,Z 1139.441,A -85,B 0,C 180,E1 21180.468,E2 21180.468} C_VEL
LIN {X 0,Y 458.485,Z 1164.834,A -85,B 0,C 180,E1 21178.228,E2 21178.228} C_VEL
LIN {X 0,Y 456.087,Z 1185.899,A -85,B 0,C 180,E1 21176.077,E2 21176.077} C_VEL
LIN {X 0,Y 453.97,Z 1205.414,A -85,B 0,C 180,E1 21173.771,E2 21173.771} C_VEL
LIN {X 0,Y 452.286,Z 1221.734,A -85,B 0,C 180,E1 21171.531,E2 21171.531} C_VEL
LIN {X 0,Y 450.954,Z 1235.709,A -85,B 0,C 180,E1 21169.293,E2 21169.293} C_VEL
LIN {X 0,Y 449.859,Z 1248.181,A -85,B 0,C 180,E1 21166.93,E2 21166.93} C_VEL
LIN {X 0,Y 449.048,Z 1259.116,A -85,B 0,C 180,E1 21164.443,E2 21164.443} C_VEL
LIN {X 0,Y 448.533,Z 1268.347,A -85,B 0,C 180,E1 21161.862,E2 21161.862} C_VEL
LIN {X 0,Y 448.241,Z 1275.36,A -85,B 0,C 180,E1 21159.373,E2 21159.373} C_VEL
LIN {X 0,Y 448.137,Z 1280.76,A -85,B 0,C 180,E1 21156.793,E2 21156.793} C_VEL
LIN {X 0,Y 448.123,Z 1284.507,A -85,B 0,C 180,E1 21154.14,E2 21154.14} C_VEL
LIN {X 0,Y 448.137,Z 1286.483,A -85,B 0,C 180,E1 21151.536,E2 21151.536} C_VEL
LIN {X 0,Y 448.143,Z 1286.73,A -85,B 0,C 180,E1 21148.979,E2 21148.979} C_VEL
LIN {X 0,Y 448.108,Z 1285.307,A -85,B 0,C 180,E1 21146.292,E2 21146.292} C_VEL
LIN {X 0,Y 448.099,Z 1282.373,A -85,B 0,C 180,E1 21143.725,E2 21143.725} C_VEL
LIN {X 0,Y 448.168,Z 1277.564,A -85,B 0,C 180,E1 21141.017,E2 21141.017} C_VEL
LIN {X 0,Y 448.468,Z 1270.655,A -85,B 0,C 180,E1 21138.165,E2 21138.165} C_VEL
LIN {X 0,Y 449.052,Z 1262.141,A -85,B 0,C 180,E1 21135.429,E2 21135.429} C_VEL
LIN {X 0,Y 450.033,Z 1251.695,A -85,B 0,C 180,E1 21132.681,E2 21132.681} C_VEL
LIN {X 0,Y 451.523,Z 1239.093,A -85,B 0,C 180,E1 21129.927,E2 21129.927} C_VEL
LIN {X 0,Y 453.48,Z 1224.957,A -85,B 0,C 180,E1 21127.305,E2 21127.305} C_VEL
LIN {X 0,Y 456.027,Z 1208.471,A -85,B 0,C 180,E1 21124.69,E2 21124.69} C_VEL
LIN {X 0,Y 459.194,Z 1189.636,A -85,B 0,C 180,E1 21122.137,E2 21122.137} C_VEL
LIN {X 0,Y 462.572,Z 1170.489,A -85,B 0,C 180,E1 21119.904,E2 21119.904} C_VEL
LIN {X 0,Y 466.386,Z 1149.679,A -85,B 0,C 180,E1 21117.81,E2 21117.81} C_VEL
LIN {X 0,Y 470.224,Z 1128.797,A -85,B 0,C 180,E1 21115.999,E2 21115.999} C_VEL
LIN {X 0,Y 474.659,Z 1105.08,A -85,B 0,C 180,E1 21114.23,E2 21114.23} C_VEL
LIN {X 0,Y 478.575,Z 1083.455,A -85,B 0,C 180,E1 21112.86,E2 21112.86} C_VEL
LIN {X 0,Y 483.178,Z 1057.339,A -85,B 0,C 180,E1 21111.475,E2 21111.475} C_VEL
LIN {X 0,Y 487.152,Z 1033.618,A -85,B 0,C 180,E1 21110.45,E2 21110.45} C_VEL
LIN {X 0,Y 490.985,Z 1007.93,A -85,B 0,C 180,E1 21109.57,E2 21109.57} C_VEL
LIN {X 0,Y 493.997,Z 982.476,A -85,B 0,C 180,E1 21108.869,E2 21108.869} C_VEL
LIN {X 0,Y 496.862,Z 960.778,A -85,B 0,C 180,E1 21108.491,E2 21108.491} C_VEL
LIN {X 0,Y 499.237,Z 946.56,A -85,B 0,C 180,E1 21108.315,E2 21108.315} C_VEL
LIN {X 0,Y 491.133,Z 931.148,A -85,B 0,C 180,E1 21107.16,E2 21107.16} C_VEL
LIN {X 0,Y 486.452,Z 912.724,A -85,B 0,C 180,E1 21104.915,E2 21104.915} C_VEL
LIN {X 0,Y 484.2,Z 893.299,A -85,B 0,C 180,E1 21102.683,E2 21102.683} C_VEL
LIN {X 0,Y 484.34,Z 871.533,A -85,B 0,C 180,E1 21100.339,E2 21100.339} C_VEL
LIN {X 0,Y 487.585,Z 843.867,A -85,B 0,C 180,E1 21097.565,E2 21097.565} C_VEL
LIN {X 0,Y 492.886,Z 809.153,A -85,B 0,C 180,E1 21094.142,E2 21094.142} C_VEL
LIN {X 0,Y 498.259,Z 775.046,A -85,B 0,C 180,E1 21090.712,E2 21090.712} C_VEL
LIN {X 0,Y 502.362,Z 748.921,A -85,B 0,C 180,E1 21088.017,E2 21088.017} C_VEL
LIN {X 0,Y 494.938,Z 730.047,A -85,B 0,C 180,E1 21084.72,E2 21084.72} C_VEL
LIN {X 0,Y 487.949,Z 713.018,A -85,B 0,C 180,E1 21081.519,E2 21081.519} C_VEL
LIN {X 0,Y 480.716,Z 696.225,A -85,B 0,C 180,E1 21078.1,E2 21078.1} C_VEL
LIN {X 0,Y 474.4,Z 682.326,A -85,B 0,C 180,E1 21075.025,E2 21075.025} C_VEL
LIN {X 0,Y 468.828,Z 670.324,A -85,B 0,C 180,E1 21072.189,E2 21072.189} C_VEL
LIN {X 0,Y 463.201,Z 658.481,A -85,B 0,C 180,E1 21069.192,E2 21069.192} C_VEL
LIN {X 0,Y 458.527,Z 649.088,A -85,B 0,C 180,E1 21066.637,E2 21066.637} C_VEL
LIN {X 0,Y 456.412,Z 644.755,A -85,B 0,C 180,E1 21065.405,E2 21065.405} C_VEL
LIN {X 0,Y 454.253,Z 640.445,A -85,B 0,C 180,E1 21064.166,E2 21064.166} C_VEL
LIN {X 0,Y 452.243,Z 636.206,A -85,B 0,C 180,E1 21062.915,E2 21062.915} C_VEL
LIN {X 0,Y 450.516,Z 632.981,A -85,B 0,C 180,E1 21061.908,E2 21061.908} C_VEL
LIN {X 0,Y 450.299,Z 631.881,A -85,B 0,C 180,E1 21061.591,E2 21061.591} C_VEL
LIN {X 0,Y 450.286,Z 631.882,A -85,B 0,C 180,E1 21057.964,E2 21057.964} C_VEL
LIN {X 0,Y 450.299,Z 631.891,A -85,B 0,C 180,E1 21054.265,E2 21054.265} C_VEL
LIN {X 0,Y 450.287,Z 631.886,A -85,B 0,C 180,E1 21050.542,E2 21050.542} C_VEL
LIN {X 0,Y 450.298,Z 631.878,A -85,B 0,C 180,E1 21046.779,E2 21046.779} C_VEL
LIN {X 0,Y 450.291,Z 631.88,A -85,B 0,C 180,E1 21043.089,E2 21043.089} C_VEL
LIN {X 0,Y 450.291,Z 631.881,A -85,B 0,C 180,E1 21039.461,E2 21039.461} C_VEL
LIN {X 0,Y 450.292,Z 631.882,A -85,B 0,C 180,E1 21035.745,E2 21035.745} C_VEL
LIN {X 0,Y 450.304,Z 631.88,A -85,B 0,C 180,E1 21031.917,E2 21031.917} C_VEL
LIN {X 0,Y 450.295,Z 631.883,A -85,B 0,C 180,E1 21028.097,E2 21028.097} C_VEL
LIN {X 0,Y 450.289,Z 631.879,A -85,B 0,C 180,E1 21024.359,E2 21024.359} C_VEL
LIN {X 0,Y 450.302,Z 631.881,A -85,B 0,C 180,E1 21020.596,E2 21020.596} C_VEL
LIN {X 0,Y 450.287,Z 631.842,A -85,B 0,C 180,E1 21016.848,E2 21016.848} C_VEL
LIN {X 0,Y 450.3,Z 631.913,A -85,B 0,C 180,E1 21013.228,E2 21013.228} C_VEL
LIN {X 0,Y 451.502,Z 635.201,A -85,B 0,C 180,E1 21012.831,E2 21012.831} C_VEL
LIN {X 0,Y 458.987,Z 652.469,A -85,B 0,C 180,E1 21010.642,E2 21010.642} C_VEL
LIN {X 0,Y 466.158,Z 671.62,A -85,B 0,C 180,E1 21008.373,E2 21008.373} C_VEL
LIN {X 0,Y 472.71,Z 692.232,A -85,B 0,C 180,E1 21006.097,E2 21006.097} C_VEL
LIN {X 0,Y 473.474,Z 695.101,A -85,B 0,C 180,E1 21005.798,E2 21005.798} C_VEL
LIN {X 0,Y 470.604,Z 739.855,A -85,B 0,C 180,E1 21002.26,E2 21002.26} C_VEL
LIN {X 0,Y 467.645,Z 787.299,A -85,B 0,C 180,E1 20998.537,E2 20998.537} C_VEL
LIN {X 0,Y 465.055,Z 835.516,A -85,B 0,C 180,E1 20994.862,E2 20994.862} C_VEL
LIN {X 0,Y 464.245,Z 856.863,A -85,B 0,C 180,E1 20993.331,E2 20993.331} C_VEL
LIN {X 0,Y 464.832,Z 864.324,A -85,B 0,C 180,E1 20993.173,E2 20993.173} C_VEL
LIN {X 0,Y 461.761,Z 1024.607,A -85,B 0,C 180,E1 20990.662,E2 20990.662} C_VEL
LIN {X 0,Y 461.39,Z 1042.464,A -85,B 0,C 180,E1 20990.176,E2 20990.176} C_VEL
LIN {X 0,Y 460.719,Z 1058.506,A -85,B 0,C 180,E1 20989.523,E2 20989.523} C_VEL
LIN {X 0,Y 459.719,Z 1074.411,A -85,B 0,C 180,E1 20988.644,E2 20988.644} C_VEL
LIN {X 0,Y 458.428,Z 1090.17,A -85,B 0,C 180,E1 20987.515,E2 20987.515} C_VEL
LIN {X 0,Y 457.007,Z 1104.784,A -85,B 0,C 180,E1 20986.196,E2 20986.196} C_VEL
LIN {X 0,Y 455.566,Z 1117.694,A -85,B 0,C 180,E1 20984.748,E2 20984.748} C_VEL
LIN {X 0,Y 454.123,Z 1129.548,A -85,B 0,C 180,E1 20983.106,E2 20983.106} C_VEL
LIN {X 0,Y 452.806,Z 1139.938,A -85,B 0,C 180,E1 20981.332,E2 20981.332} C_VEL
LIN {X 0,Y 451.668,Z 1148.903,A -85,B 0,C 180,E1 20979.427,E2 20979.427} C_VEL
LIN {X 0,Y 450.747,Z 1156.367,A -85,B 0,C 180,E1 20977.39,E2 20977.39} C_VEL
LIN {X 0,Y 450.067,Z 1162.264,A -85,B 0,C 180,E1 20975.224,E2 20975.224} C_VEL
LIN {X 0,Y 449.638,Z 1166.339,A -85,B 0,C 180,E1 20973.058,E2 20973.058} C_VEL
LIN {X 0,Y 449.416,Z 1168.815,A -85,B 0,C 180,E1 20970.763,E2 20970.763} C_VEL
LIN {X 0,Y 449.371,Z 1169.412,A -85,B 0,C 180,E1 20968.468,E2 20968.468} C_VEL
LIN {X 0,Y 449.398,Z 1169.264,A -85,B 0,C 180,E1 20967.759,E2 20967.759} C_VEL
LIN {X 0,Y 448.46,Z 1168.869,A -85,B 0,C 180,E1 20966.776,E2 20966.776} C_VEL
LIN {X 0,Y 443.623,Z 1167.374,A -85,B 0,C 180,E1 20964.718,E2 20964.718} C_VEL
LIN {X 0,Y 442.079,Z 1165.841,A -85,B 0,C 180,E1 20963.598,E2 20963.598} C_VEL
LIN {X 0,Y 442.053,Z 1165.325,A -85,B 0,C 180,E1 20963.317,E2 20963.317} C_VEL
LIN {X 0,Y 442.745,Z 1160.093,A -85,B 0,C 180,E1 20961.033,E2 20961.033} C_VEL
LIN {X 0,Y 443.66,Z 1153.477,A -85,B 0,C 180,E1 20958.954,E2 20958.954} C_VEL
LIN {X 0,Y 444.886,Z 1144.814,A -85,B 0,C 180,E1 20956.878,E2 20956.878} C_VEL
LIN {X 0,Y 446.351,Z 1134.559,A -85,B 0,C 180,E1 20954.937,E2 20954.937} C_VEL
LIN {X 0,Y 447.867,Z 1123.558,A -85,B 0,C 180,E1 20953.26,E2 20953.26} C_VEL
LIN {X 0,Y 449.507,Z 1110.46,A -85,B 0,C 180,E1 20951.652,E2 20951.652} C_VEL
LIN {X 0,Y 451.11,Z 1096.228,A -85,B 0,C 180,E1 20950.242,E2 20950.242} C_VEL
LIN {X 0,Y 452.499,Z 1081.746,A -85,B 0,C 180,E1 20949.091,E2 20949.091} C_VEL
LIN {X 0,Y 453.707,Z 1065.717,A -85,B 0,C 180,E1 20948.097,E2 20948.097} C_VEL
LIN {X 0,Y 454.626,Z 1048.519,A -85,B 0,C 180,E1 20947.302,E2 20947.302} C_VEL
LIN {X 0,Y 455.171,Z 1030.977,A -85,B 0,C 180,E1 20946.741,E2 20946.741} C_VEL
LIN {X 0,Y 455.475,Z 1002.886,A -85,B 0,C 180,E1 20946.233,E2 20946.233} C_VEL
LIN {X 0,Y 458.408,Z 862.048,A -85,B 0,C 180,E1 20944.006,E2 20944.006} C_VEL
LIN {X 0,Y 457.844,Z 856.714,A -85,B 0,C 180,E1 20943.843,E2 20943.843} C_VEL
LIN {X 0,Y 460.155,Z 811.595,A -85,B 0,C 180,E1 20940.444,E2 20940.444} C_VEL
LIN {X 0,Y 463.178,Z 764.519,A -85,B 0,C 180,E1 20936.746,E2 20936.746} C_VEL
LIN {X 0,Y 466.257,Z 719.694,A -85,B 0,C 180,E1 20933.172,E2 20933.172} C_VEL
LIN {X 0,Y 467.538,Z 699.012,A -85,B 0,C 180,E1 20931.511,E2 20931.511} C_VEL
LIN {X 0,Y 461.109,Z 678.625,A -85,B 0,C 180,E1 20929.182,E2 20929.182} C_VEL
LIN {X 0,Y 456.818,Z 666.726,A -85,B 0,C 180,E1 20927.737,E2 20927.737} C_VEL
LIN {X 0,Y 458.666,Z 667.539,A -85,B 0,C 180,E1 20927.482,E2 20927.482} C_VEL
LIN {X 0,Y 460.632,Z 667.419,A -85,B 0,C 180,E1 20927.242,E2 20927.242} C_VEL
LIN {X 0,Y 476.353,Z 689.24,A -85,B 0,C 180,E1 20924.699,E2 20924.699} C_VEL
LIN {X 0,Y 494.315,Z 715.668,A -85,B 0,C 180,E1 20922.042,E2 20922.042} C_VEL
LIN {X 0,Y 496.063,Z 718.731,A -85,B 0,C 180,E1 20921.783,E2 20921.783} C_VEL
LIN {X 0,Y 478.647,Z 975.997,A -85,B 0,C 180,E1 20916.571,E2 20916.571} C_VEL
LIN {X 0,Y 476.854,Z 999.63,A -85,B 0,C 180,E1 20915.868,E2 20915.868} C_VEL
LIN {X 0,Y 474.556,Z 1022.561,A -85,B 0,C 180,E1 20914.967,E2 20914.967} C_VEL
LIN {X 0,Y 471.984,Z 1043.518,A -85,B 0,C 180,E1 20913.933,E2 20913.933} C_VEL
LIN {X 0,Y 468.901,Z 1064.823,A -85,B 0,C 180,E1 20912.65,E2 20912.65} C_VEL
LIN {X 0,Y 465.478,Z 1086.119,A -85,B 0,C 180,E1 20911.106,E2 20911.106} C_VEL
LIN {X 0,Y 462.033,Z 1105.693,A -85,B 0,C 180,E1 20909.423,E2 20909.423} C_VEL
LIN {X 0,Y 458.488,Z 1124.162,A -85,B 0,C 180,E1 20907.538,E2 20907.538} C_VEL
LIN {X 0,Y 454.977,Z 1141.955,A -85,B 0,C 180,E1 20905.41,E2 20905.41} C_VEL
LIN {X 0,Y 451.803,Z 1157.801,A -85,B 0,C 180,E1 20903.2,E2 20903.2} C_VEL
LIN {X 0,Y 448.97,Z 1171.964,A -85,B 0,C 180,E1 20900.875,E2 20900.875} C_VEL
LIN {X 0,Y 446.357,Z 1185.461,A -85,B 0,C 180,E1 20898.277,E2 20898.277} C_VEL
LIN {X 0,Y 444.318,Z 1196.973,A -85,B 0,C 180,E1 20895.667,E2 20895.667} C_VEL
LIN {X 0,Y 442.693,Z 1207.015,A -85,B 0,C 180,E1 20892.921,E2 20892.921} C_VEL
LIN {X 0,Y 441.525,Z 1215.633,A -85,B 0,C 180,E1 20890.042,E2 20890.042} C_VEL
LIN {X 0,Y 440.827,Z 1222.262,A -85,B 0,C 180,E1 20887.297,E2 20887.297} C_VEL
LIN {X 0,Y 440.405,Z 1227.42,A -85,B 0,C 180,E1 20884.427,E2 20884.427} C_VEL
LIN {X 0,Y 440.223,Z 1231.202,A -85,B 0,C 180,E1 20881.432,E2 20881.432} C_VEL
LIN {X 0,Y 440.175,Z 1233.106,A -85,B 0,C 180,E1 20878.829,E2 20878.829} C_VEL
LIN {X 0,Y 440.192,Z 1233.765,A -85,B 0,C 180,E1 20875.832,E2 20875.832} C_VEL
LIN {X 0,Y 440.282,Z 1232.974,A -85,B 0,C 180,E1 20873.087,E2 20873.087} C_VEL
LIN {X 0,Y 440.51,Z 1230.57,A -85,B 0,C 180,E1 20870.198,E2 20870.198} C_VEL
LIN {X 0,Y 440.974,Z 1226.693,A -85,B 0,C 180,E1 20867.294,E2 20867.294} C_VEL
LIN {X 0,Y 441.762,Z 1221.443,A -85,B 0,C 180,E1 20864.509,E2 20864.509} C_VEL
LIN {X 0,Y 443.057,Z 1214.229,A -85,B 0,C 180,E1 20861.582,E2 20861.582} C_VEL
LIN {X 0,Y 444.861,Z 1205.64,A -85,B 0,C 180,E1 20858.785,E2 20858.785} C_VEL
LIN {X 0,Y 447.277,Z 1195.148,A -85,B 0,C 180,E1 20855.992,E2 20855.992} C_VEL
LIN {X 0,Y 450.02,Z 1183.671,A -85,B 0,C 180,E1 20853.474,E2 20853.474} C_VEL
LIN {X 0,Y 453.352,Z 1170.164,A -85,B 0,C 180,E1 20850.973,E2 20850.973} C_VEL
LIN {X 0,Y 456.829,Z 1156.014,A -85,B 0,C 180,E1 20848.752,E2 20848.752} C_VEL
LIN {X 0,Y 460.552,Z 1140.435,A -85,B 0,C 180,E1 20846.682,E2 20846.682} C_VEL
LIN {X 0,Y 464.232,Z 1123.79,A -85,B 0,C 180,E1 20844.819,E2 20844.819} C_VEL
LIN {X 0,Y 467.791,Z 1106.301,A -85,B 0,C 180,E1 20843.161,E2 20843.161} C_VEL
LIN {X 0,Y 471.121,Z 1088.052,A -85,B 0,C 180,E1 20841.703,E2 20841.703} C_VEL
LIN {X 0,Y 474.108,Z 1069.002,A -85,B 0,C 180,E1 20840.438,E2 20840.438} C_VEL
LIN {X 0,Y 476.764,Z 1048.491,A -85,B 0,C 180,E1 20839.328,E2 20839.328} C_VEL
LIN {X 0,Y 478.886,Z 1026.871,A -85,B 0,C 180,E1 20838.412,E2 20838.412} C_VEL
LIN {X 0,Y 480.364,Z 1004.889,A -85,B 0,C 180,E1 20837.707,E2 20837.707} C_VEL
LIN {X 0,Y 483.328,Z 972.35,A -85,B 0,C 180,E1 20836.829,E2 20836.829} C_VEL
LIN {X 0,Y 488.833,Z 936.196,A -85,B 0,C 180,E1 20835.87,E2 20835.87} C_VEL
LIN {X 0,Y 496.863,Z 897.588,A -85,B 0,C 180,E1 20834.795,E2 20834.795} C_VEL
LIN {X 0,Y 497.591,Z 894.436,A -85,B 0,C 180,E1 20834.695,E2 20834.695} C_VEL
LIN {X 0,Y 495.081,Z 905.3,A -85,B 0,C 180,E1 20833.429,E2 20833.429} C_VEL
LIN {X 0,Y 494.607,Z 917.29,A -85,B 0,C 180,E1 20832.104,E2 20832.104} C_VEL
LIN {X 0,Y 495.345,Z 924.791,A -85,B 0,C 180,E1 20831.3,E2 20831.3} C_VEL
LIN {X 0,Y 489.655,Z 944.349,A -85,B 0,C 180,E1 20831.172,E2 20831.172} C_VEL
LIN {X 0,Y 484.586,Z 963.592,A -85,B 0,C 180,E1 20830.813,E2 20830.813} C_VEL
LIN {X 0,Y 480.443,Z 981.572,A -85,B 0,C 180,E1 20830.258,E2 20830.258} C_VEL
LIN {X 0,Y 473.452,Z 1017.993,A -85,B 0,C 180,E1 20828.693,E2 20828.693} C_VEL
LIN {X 0,Y 467.534,Z 1051.074,A -85,B 0,C 180,E1 20827.017,E2 20827.017} C_VEL
LIN {X 0,Y 462.2,Z 1083.98,A -85,B 0,C 180,E1 20825.057,E2 20825.057} C_VEL
LIN {X 0,Y 457.863,Z 1113.608,A -85,B 0,C 180,E1 20823.008,E2 20823.008} C_VEL
LIN {X 0,Y 454.113,Z 1141.4,A -85,B 0,C 180,E1 20820.801,E2 20820.801} C_VEL
LIN {X 0,Y 450.976,Z 1166.003,A -85,B 0,C 180,E1 20818.543,E2 20818.543} C_VEL
LIN {X 0,Y 448.29,Z 1188.111,A -85,B 0,C 180,E1 20816.209,E2 20816.209} C_VEL
LIN {X 0,Y 446.156,Z 1206.7,A -85,B 0,C 180,E1 20813.933,E2 20813.933} C_VEL
LIN {X 0,Y 444.393,Z 1222.705,A -85,B 0,C 180,E1 20811.656,E2 20811.656} C_VEL
LIN {X 0,Y 442.939,Z 1237.167,A -85,B 0,C 180,E1 20809.245,E2 20809.245} C_VEL
LIN {X 0,Y 441.814,Z 1249.573,A -85,B 0,C 180,E1 20806.8,E2 20806.8} C_VEL
LIN {X 0,Y 441.013,Z 1260.085,A -85,B 0,C 180,E1 20804.309,E2 20804.309} C_VEL
LIN {X 0,Y 440.517,Z 1268.685,A -85,B 0,C 180,E1 20801.789,E2 20801.789} C_VEL
LIN {X 0,Y 440.234,Z 1275.428,A -85,B 0,C 180,E1 20799.282,E2 20799.282} C_VEL
LIN {X 0,Y 440.136,Z 1280.706,A -85,B 0,C 180,E1 20796.655,E2 20796.655} C_VEL
LIN {X 0,Y 440.133,Z 1284.225,A -85,B 0,C 180,E1 20794.04,E2 20794.04} C_VEL
LIN {X 0,Y 440.153,Z 1286.012,A -85,B 0,C 180,E1 20791.434,E2 20791.434} C_VEL
LIN {X 0,Y 440.155,Z 1286.166,A -85,B 0,C 180,E1 20788.83,E2 20788.83} C_VEL
LIN {X 0,Y 440.124,Z 1284.734,A -85,B 0,C 180,E1 20786.224,E2 20786.224} C_VEL
LIN {X 0,Y 440.108,Z 1281.743,A -85,B 0,C 180,E1 20783.61,E2 20783.61} C_VEL
LIN {X 0,Y 440.186,Z 1276.839,A -85,B 0,C 180,E1 20780.853,E2 20780.853} C_VEL
LIN {X 0,Y 440.49,Z 1270.127,A -85,B 0,C 180,E1 20778.057,E2 20778.057} C_VEL
LIN {X 0,Y 441.087,Z 1261.651,A -85,B 0,C 180,E1 20775.294,E2 20775.294} C_VEL
LIN {X 0,Y 442.105,Z 1251.165,A -85,B 0,C 180,E1 20772.496,E2 20772.496} C_VEL
LIN {X 0,Y 443.561,Z 1239.163,A -85,B 0,C 180,E1 20769.827,E2 20769.827} C_VEL
LIN {X 0,Y 445.564,Z 1225.103,A -85,B 0,C 180,E1 20767.158,E2 20767.158} C_VEL
LIN {X 0,Y 448.318,Z 1207.77,A -85,B 0,C 180,E1 20764.365,E2 20764.365} C_VEL
LIN {X 0,Y 451.56,Z 1189.098,A -85,B 0,C 180,E1 20761.799,E2 20761.799} C_VEL
LIN {X 0,Y 455.103,Z 1169.687,A -85,B 0,C 180,E1 20759.504,E2 20759.504} C_VEL
LIN {X 0,Y 459.043,Z 1148.869,A -85,B 0,C 180,E1 20757.38,E2 20757.38} C_VEL
LIN {X 0,Y 463.007,Z 1127.979,A -85,B 0,C 180,E1 20755.545,E2 20755.545} C_VEL
LIN {X 0,Y 467.577,Z 1104.335,A -85,B 0,C 180,E1 20753.755,E2 20753.755} C_VEL
LIN {X 0,Y 471.739,Z 1082.065,A -85,B 0,C 180,E1 20752.326,E2 20752.326} C_VEL
LIN {X 0,Y 476.553,Z 1055.673,A -85,B 0,C 180,E1 20750.916,E2 20750.916} C_VEL
LIN {X 0,Y 480.522,Z 1032.666,A -85,B 0,C 180,E1 20749.911,E2 20749.911} C_VEL
LIN {X 0,Y 484.556,Z 1006.413,A -85,B 0,C 180,E1 20748.997,E2 20748.997} C_VEL
LIN {X 0,Y 487.715,Z 980.53,A -85,B 0,C 180,E1 20748.28,E2 20748.28} C_VEL
LIN {X 0,Y 490.779,Z 958.695,A -85,B 0,C 180,E1 20747.908,E2 20747.908} C_VEL
LIN {X 0,Y 492.309,Z 949.217,A -85,B 0,C 180,E1 20747.785,E2 20747.785} C_VEL
LIN {X 0,Y 482.926,Z 930.467,A -85,B 0,C 180,E1 20746.399,E2 20746.399} C_VEL
LIN {X 0,Y 482.112,Z 928.168,A -85,B 0,C 180,E1 20746.199,E2 20746.199} C_VEL
LIN {X 0,Y 478.32,Z 909.546,A -85,B 0,C 180,E1 20743.949,E2 20743.949} C_VEL
LIN {X 0,Y 476.881,Z 889.442,A -85,B 0,C 180,E1 20741.657,E2 20741.657} C_VEL
LIN {X 0,Y 477.942,Z 866.249,A -85,B 0,C 180,E1 20739.184,E2 20739.184} C_VEL
LIN {X 0,Y 484.976,Z 818.778,A -85,B 0,C 180,E1 20734.447,E2 20734.447} C_VEL
LIN {X 0,Y 490.414,Z 785.162,A -85,B 0,C 180,E1 20731.053,E2 20731.053} C_VEL
LIN {X 0,Y 495.748,Z 752.928,A -85,B 0,C 180,E1 20727.727,E2 20727.727} C_VEL
LIN {X 0,Y 488.974,Z 735.449,A -85,B 0,C 180,E1 20724.655,E2 20724.655} C_VEL
LIN {X 0,Y 482.003,Z 718.333,A -85,B 0,C 180,E1 20721.414,E2 20721.414} C_VEL
LIN {X 0,Y 475.168,Z 702.394,A -85,B 0,C 180,E1 20718.146,E2 20718.146} C_VEL
LIN {X 0,Y 468.732,Z 688.004,A -85,B 0,C 180,E1 20714.958,E2 20714.958} C_VEL
LIN {X 0,Y 462.083,Z 673.47,A -85,B 0,C 180,E1 20711.483,E2 20711.483} C_VEL
LIN {X 0,Y 455.59,Z 659.868,A -85,B 0,C 180,E1 20707.948,E2 20707.948} C_VEL
LIN {X 0,Y 450.728,Z 650.221,A -85,B 0,C 180,E1 20705.219,E2 20705.219} C_VEL
LIN {X 0,Y 448.568,Z 645.918,A -85,B 0,C 180,E1 20703.962,E2 20703.962} C_VEL
LIN {X 0,Y 446.543,Z 641.712,A -85,B 0,C 180,E1 20702.695,E2 20702.695} C_VEL
LIN {X 0,Y 444.748,Z 637.829,A -85,B 0,C 180,E1 20701.546,E2 20701.546} C_VEL
LIN {X 0,Y 442.577,Z 633.997,A -85,B 0,C 180,E1 20700.259,E2 20700.259} C_VEL
LIN {X 0,Y 442.347,Z 632.879,A -85,B 0,C 180,E1 20699.935,E2 20699.935} C_VEL
LIN {X 0,Y 442.353,Z 632.87,A -85,B 0,C 180,E1 20696.112,E2 20696.112} C_VEL
LIN {X 0,Y 442.362,Z 632.868,A -85,B 0,C 180,E1 20692.336,E2 20692.336} C_VEL
LIN {X 0,Y 442.349,Z 632.879,A -85,B 0,C 180,E1 20688.526,E2 20688.526} C_VEL
LIN {X 0,Y 442.369,Z 632.88,A -85,B 0,C 180,E1 20684.799,E2 20684.799} C_VEL
LIN {X 0,Y 442.364,Z 632.874,A -85,B 0,C 180,E1 20680.868,E2 20680.868} C_VEL
LIN {X 0,Y 442.349,Z 632.872,A -85,B 0,C 180,E1 20677.121,E2 20677.121} C_VEL
LIN {X 0,Y 442.356,Z 632.867,A -85,B 0,C 180,E1 20673.413,E2 20673.413} C_VEL
LIN {X 0,Y 442.352,Z 632.869,A -85,B 0,C 180,E1 20669.704,E2 20669.704} C_VEL
LIN {X 0,Y 442.362,Z 632.867,A -85,B 0,C 180,E1 20665.817,E2 20665.817} C_VEL
LIN {X 0,Y 442.363,Z 632.869,A -85,B 0,C 180,E1 20662.061,E2 20662.061} C_VEL
LIN {X 0,Y 442.348,Z 632.856,A -85,B 0,C 180,E1 20658.351,E2 20658.351} C_VEL
